    |   movel([0.402308, -0.603940, -2.826285, -1.282164, 1.570796, 1.973104],accel_mss,speed_ms,0,blend_radius_m)
    |   movel([0.405930, -0.602202, -2.826422, -1.283765, 1.570796, 1.976727],accel_mss,speed_ms,0,blend_radius_m)
    |   movel([0.409236, -0.601189, -2.826501, -1.284699, 1.570796, 1.980032],accel_mss,speed_ms,0,blend_radius_m)
    |   movel([0.412170, -0.600886, -2.826525, -1.284978, 1.570796, 1.982967],accel_mss,speed_ms,0,blend_radius_m)
    |   movel([0.414677, -0.601290, -2.826494, -1.284605, 1.570796, 1.985473],accel_mss,speed_ms,0,blend_radius_m)
    |   movel([0.416713, -0.602370, -2.826409, -1.283610, 1.570796, 1.987509],accel_mss,speed_ms,0,blend_radius_m)
    |   movel([0.418227, -0.604116, -2.826271, -1.282003, 1.570796, 1.989024],accel_mss,speed_ms,0,blend_radius_m)
    |   movel([0.419169, -0.606504, -2.826080, -1.279805, 1.570796, 1.989965],accel_mss,speed_ms,0,blend_radius_m)
    |   movel([0.419507, -0.609503, -2.825837, -1.277049, 1.570796, 1.990303],accel_mss,speed_ms,0,blend_radius_m)
    |   speed_ms = 0.005
    |   movel([0.419507, -0.603604, -2.819016, -1.289768, 1.570796, 1.990303],accel_mss,speed_ms,0,blend_radius_m)
    |   speed_ms = 0.040
    |   movel([0.367133, -0.571000, -2.821459, -1.319930, 1.570796, 1.937929],accel_mss,speed_ms,0,blend_radius_m)
    |   speed_ms = 0.005
    |   movel([0.367133, -0.576329, -2.828331, -1.307729, 1.570796, 1.937929],accel_mss,speed_ms,0,blend_radius_m)
    |   speed_ms = 0.025
    |   movel([0.368594, -0.576617, -2.828311, -1.307461, 1.570796, 1.939390],accel_mss,speed_ms,0,blend_radius_m)
    |   movel([0.369540, -0.577566, -2.828246, -1.306577, 1.570796, 1.940337],accel_mss,speed_ms,0,blend_radius_m)
    |   movel([0.369616, -0.578487, -2.828182, -1.305720, 1.570796, 1.940412],accel_mss,speed_ms,0,blend_radius_m)
    |   movel([0.369337, -0.579700, -2.828097, -1.304592, 1.570796, 1.940133],accel_mss,speed_ms,0,blend_radius_m)
    |   movel([0.368717, -0.581070, -2.828000, -1.303319, 1.570796, 1.939513],accel_mss,speed_ms,0,blend_radius_m)
    |   movel([0.367757, -0.582464, -2.827901, -1.302024, 1.570796, 1.938554],accel_mss,speed_ms,0,blend_radius_m)
    |   movel([0.365671, -0.584790, -2.827735, -1.299864, 1.570796, 1.936467],accel_mss,speed_ms,0,blend_radius_m)
    |   movel([0.364856, -0.586105, -2.827639, -1.298645, 1.570796, 1.935652],accel_mss,speed_ms,0,blend_radius_m)
    |   movel([0.364407, -0.587333, -2.827550, -1.297506, 1.570796, 1.935203],accel_mss,speed_ms,0,blend_radius_m)
    |   movel([0.364314, -0.589341, -2.827403, -1.295646, 1.570796, 1.935110],accel_mss,speed_ms,0,blend_radius_m)
    |   movel([0.364860, -0.591067, -2.827275, -1.294047, 1.570796, 1.935656],accel_mss,speed_ms,0,blend_radius_m)
    |   movel([0.365794, -0.592354, -2.827178, -1.292856, 1.570796, 1.936590],accel_mss,speed_ms,0,blend_radius_m)
    |   movel([0.367088, -0.593198, -2.827115, -1.292076, 1.570796, 1.937884],accel_mss,speed_ms,0,blend_radius_m)
    |   movel([0.368715, -0.593567, -2.827087, -1.291734, 1.570796, 1.939512],accel_mss,speed_ms,0,blend_radius_m)
    |   movel([0.366876, -0.596507, -2.826864, -1.289018, 1.570796, 1.937672],accel_mss,speed_ms,0,blend_radius_m)
    |   movel([0.365400, -0.599354, -2.826644, -1.286390, 1.570796, 1.936197],accel_mss,speed_ms,0,blend_radius_m)
    |   movel([0.364245, -0.602108, -2.826429, -1.283852, 1.570796, 1.935041],accel_mss,speed_ms,0,blend_radius_m)
    |   movel([0.363369, -0.604758, -2.826220, -1.281412, 1.570796, 1.934166],accel_mss,speed_ms,0,blend_radius_m)
    |   movel([0.362308, -0.609715, -2.825820, -1.276854, 1.570796, 1.933104],accel_mss,speed_ms,0,blend_radius_m)
    |   movel([0.361927, -0.614158, -2.825454, -1.272778, 1.570796, 1.932724],accel_mss,speed_ms,0,blend_radius_m)
    |   movel([0.361646, -0.618378, -2.825099, -1.268912, 1.570796, 1.932442],accel_mss,speed_ms,0,blend_radius_m)
    |   movel([0.361180, -0.620703, -2.824900, -1.266786, 1.570796, 1.931976],accel_mss,speed_ms,0,blend_radius_m)
    |   movel([0.360296, -0.623272, -2.824678, -1.264439, 1.570796, 1.931092],accel_mss,speed_ms,0,blend_radius_m)
    |   movel([0.358808, -0.626113, -2.824430, -1.261847, 1.570796, 1.929605],accel_mss,speed_ms,0,blend_radius_m)
    |   movel([0.356822, -0.628911, -2.824182, -1.259296, 1.570796, 1.927618],accel_mss,speed_ms,0,blend_radius_m)
    |   movel([0.354611, -0.631231, -2.823974, -1.257183, 1.570796, 1.925407],accel_mss,speed_ms,0,blend_radius_m)
    |   movel([0.352461, -0.632627, -2.823848, -1.255913, 1.570796, 1.923258],accel_mss,speed_ms,0,blend_radius_m)
    |   movel([0.353015, -0.634018, -2.823722, -1.254649, 1.570796, 1.923811],accel_mss,speed_ms,0,blend_radius_m)
    |   movel([0.353232, -0.637667, -2.823387, -1.251336, 1.570796, 1.924028],accel_mss,speed_ms,0,blend_radius_m)
    |   movel([0.352907, -0.639851, -2.823184, -1.249354, 1.570796, 1.923703],accel_mss,speed_ms,0,blend_radius_m)
    |   movel([0.351453, -0.644729, -2.822723, -1.244937, 1.570796, 1.922249],accel_mss,speed_ms,0,blend_radius_m)
    |   movel([0.350339, -0.647346, -2.822472, -1.242571, 1.570796, 1.921135],accel_mss,speed_ms,0,blend_radius_m)
    |   movel([0.348974, -0.650037, -2.822211, -1.240141, 1.570796, 1.919770],accel_mss,speed_ms,0,blend_radius_m)
    |   speed_ms = 0.005
    |   movel([0.348974, -0.643483, -2.815463, -1.253443, 1.570796, 1.919770],accel_mss,speed_ms,0,blend_radius_m)
    |   speed_ms = 0.040
    |   movel([0.338843, -0.648119, -2.815009, -1.249261, 1.570796, 1.909639],accel_mss,speed_ms,0,blend_radius_m)
    |   speed_ms = 0.005
    |   movel([0.338843, -0.654746, -2.821747, -1.235896, 1.570796, 1.909639],accel_mss,speed_ms,0,blend_radius_m)
    |   speed_ms = 0.025
    |   movel([0.341191, -0.672764, -2.819888, -1.219737, 1.570796, 1.911987],accel_mss,speed_ms,0,blend_radius_m)
    |   movel([0.341193, -0.675205, -2.819625, -1.217559, 1.570796, 1.911989],accel_mss,speed_ms,0,blend_radius_m)
    |   movel([0.340796, -0.676644, -2.819469, -1.216275, 1.570796, 1.911593],accel_mss,speed_ms,0,blend_radius_m)
    |   movel([0.339964, -0.678224, -2.819297, -1.214867, 1.570796, 1.910761],accel_mss,speed_ms,0,blend_radius_m)
    |   movel([0.337481, -0.681582, -2.818928, -1.211878, 1.570796, 1.908277],accel_mss,speed_ms,0,blend_radius_m)
    |   movel([0.336864, -0.683225, -2.818746, -1.210418, 1.570796, 1.907661],accel_mss,speed_ms,0,blend_radius_m)
    |   movel([0.336819, -0.684555, -2.818597, -1.209237, 1.570796, 1.907615],accel_mss,speed_ms,0,blend_radius_m)
    |   movel([0.337450, -0.686133, -2.818420, -1.207836, 1.570796, 1.908246],accel_mss,speed_ms,0,blend_radius_m)
    |   movel([0.338671, -0.687133, -2.818307, -1.206949, 1.570796, 1.909467],accel_mss,speed_ms,0,blend_radius_m)
    |   movel([0.341481, -0.688557, -2.818146, -1.205686, 1.570796, 1.912277],accel_mss,speed_ms,0,blend_radius_m)
    |   movel([0.342858, -0.690102, -2.817970, -1.204317, 1.570796, 1.913655],accel_mss,speed_ms,0,blend_radius_m)
    |   movel([0.344241, -0.692917, -2.817646, -1.201826, 1.570796, 1.915038],accel_mss,speed_ms,0,blend_radius_m)
    |   movel([0.344493, -0.694532, -2.817459, -1.200397, 1.570796, 1.915290],accel_mss,speed_ms,0,blend_radius_m)
    |   movel([0.344236, -0.696132, -2.817273, -1.198984, 1.570796, 1.915033],accel_mss,speed_ms,0,blend_radius_m)
    |   movel([0.343860, -0.696890, -2.817184, -1.198315, 1.570796, 1.914657],accel_mss,speed_ms,0,blend_radius_m)
    |   movel([0.343290, -0.697601, -2.817101, -1.197687, 1.570796, 1.914087],accel_mss,speed_ms,0,blend_radius_m)
    |   movel([0.341482, -0.698845, -2.816954, -1.196590, 1.570796, 1.912278],accel_mss,speed_ms,0,blend_radius_m)
    |   movel([0.341411, -0.700428, -2.816767, -1.195194, 1.570796, 1.912208],accel_mss,speed_ms,0,blend_radius_m)
    |   movel([0.341805, -0.701849, -2.816597, -1.193942, 1.570796, 1.912601],accel_mss,speed_ms,0,blend_radius_m)
    |   movel([0.343551, -0.704211, -2.816314, -1.191864, 1.570796, 1.914347],accel_mss,speed_ms,0,blend_radius_m)
    |   movel([0.347880, -0.707172, -2.815955, -1.189261, 1.570796, 1.918676],accel_mss,speed_ms,0,blend_radius_m)
    |   movel([0.350537, -0.707948, -2.815861, -1.188580, 1.570796, 1.921334],accel_mss,speed_ms,0,blend_radius_m)
    |   movel([0.353591, -0.708352, -2.815812, -1.188225, 1.570796, 1.924387],accel_mss,speed_ms,0,blend_radius_m)
    |   movel([0.356222, -0.709277, -2.815698, -1.187414, 1.570796, 1.927019],accel_mss,speed_ms,0,blend_radius_m)
    |   movel([0.357125, -0.710205, -2.815584, -1.186600, 1.570796, 1.927922],accel_mss,speed_ms,0,blend_radius_m)
    |   movel([0.357618, -0.711589, -2.815414, -1.185387, 1.570796, 1.928414],accel_mss,speed_ms,0,blend_radius_m)
    |   movel([0.357593, -0.712558, -2.815293, -1.184537, 1.570796, 1.928389],accel_mss,speed_ms,0,blend_radius_m)
    |   movel([0.357273, -0.713718, -2.815149, -1.183522, 1.570796, 1.928070],accel_mss,speed_ms,0,blend_radius_m)
    |   movel([0.356670, -0.714860, -2.815006, -1.182522, 1.570796, 1.927467],accel_mss,speed_ms,0,blend_radius_m)
    |   movel([0.355782, -0.715776, -2.814892, -1.181721, 1.570796, 1.926579],accel_mss,speed_ms,0,blend_radius_m)
    |   movel([0.354440, -0.716164, -2.814843, -1.181382, 1.570796, 1.925237],accel_mss,speed_ms,0,blend_radius_m)
    |   movel([0.349203, -0.715563, -2.814918, -1.181908, 1.570796, 1.919999],accel_mss,speed_ms,0,blend_radius_m)
    |   movel([0.344633, -0.713927, -2.815123, -1.183339, 1.570796, 1.915430],accel_mss,speed_ms,0,blend_radius_m)
    |   movel([0.344030, -0.715213, -2.814962, -1.182213, 1.570796, 1.914826],accel_mss,speed_ms,0,blend_radius_m)
    |   movel([0.343689, -0.716395, -2.814814, -1.181180, 1.570796, 1.914486],accel_mss,speed_ms,0,blend_radius_m)
    |   movel([0.343697, -0.718463, -2.814553, -1.179373, 1.570796, 1.914493],accel_mss,speed_ms,0,blend_radius_m)
    |   movel([0.344441, -0.720163, -2.814337, -1.177889, 1.570796, 1.915238],accel_mss,speed_ms,0,blend_radius_m)
    |   movel([0.345698, -0.721557, -2.814158, -1.176674, 1.570796, 1.916494],accel_mss,speed_ms,0,blend_radius_m)
    |   movel([0.348943, -0.723539, -2.813903, -1.174947, 1.570796, 1.919739],accel_mss,speed_ms,0,blend_radius_m)
    |   movel([0.351761, -0.724708, -2.813752, -1.173929, 1.570796, 1.922558],accel_mss,speed_ms,0,blend_radius_m)
    |   movel([0.352666, -0.725330, -2.813672, -1.173387, 1.570796, 1.923462],accel_mss,speed_ms,0,blend_radius_m)
    |   movel([0.352850, -0.725902, -2.813597, -1.172890, 1.570796, 1.923647],accel_mss,speed_ms,0,blend_radius_m)
    |   movel([0.352704, -0.726735, -2.813489, -1.172166, 1.570796, 1.923501],accel_mss,speed_ms,0,blend_radius_m)
    |   movel([0.352198, -0.727778, -2.813352, -1.171259, 1.570796, 1.922994],accel_mss,speed_ms,0,blend_radius_m)
    |   movel([0.351586, -0.728539, -2.813253, -1.170597, 1.570796, 1.922382],accel_mss,speed_ms,0,blend_radius_m)
    |   movel([0.350182, -0.729503, -2.813126, -1.169760, 1.570796, 1.920979],accel_mss,speed_ms,0,blend_radius_m)
    |   movel([0.348239, -0.730639, -2.812976, -1.168774, 1.570796, 1.919035],accel_mss,speed_ms,0,blend_radius_m)
    |   movel([0.347795, -0.731218, -2.812899, -1.168272, 1.570796, 1.918591],accel_mss,speed_ms,0,blend_radius_m)
    |   movel([0.347475, -0.732077, -2.812785, -1.167527, 1.570796, 1.918272],accel_mss,speed_ms,0,blend_radius_m)
    |   movel([0.347450, -0.732856, -2.812681, -1.166851, 1.570796, 1.918246],accel_mss,speed_ms,0,blend_radius_m)
    |   movel([0.348020, -0.734168, -2.812506, -1.165715, 1.570796, 1.918817],accel_mss,speed_ms,0,blend_radius_m)
    |   movel([0.349767, -0.735900, -2.812273, -1.164216, 1.570796, 1.920563],accel_mss,speed_ms,0,blend_radius_m)
    |   movel([0.358098, -0.742064, -2.811434, -1.158891, 1.570796, 1.928895],accel_mss,speed_ms,0,blend_radius_m)
    |   movel([0.358752, -0.742913, -2.811317, -1.158158, 1.570796, 1.929548],accel_mss,speed_ms,0,blend_radius_m)
    |   movel([0.359088, -0.744094, -2.811154, -1.157141, 1.570796, 1.929884],accel_mss,speed_ms,0,blend_radius_m)
    |   movel([0.358896, -0.745566, -2.810950, -1.155873, 1.570796, 1.929692],accel_mss,speed_ms,0,blend_radius_m)
    |   movel([0.357966, -0.747279, -2.810711, -1.154400, 1.570796, 1.928763],accel_mss,speed_ms,0,blend_radius_m)
    |   movel([0.356641, -0.748610, -2.810524, -1.153255, 1.570796, 1.927438],accel_mss,speed_ms,0,blend_radius_m)
    |   movel([0.355296, -0.749300, -2.810427, -1.152662, 1.570796, 1.926093],accel_mss,speed_ms,0,blend_radius_m)
    |   movel([0.354031, -0.749499, -2.810399, -1.152491, 1.570796, 1.924828],accel_mss,speed_ms,0,blend_radius_m)
    |   movel([0.352947, -0.749370, -2.810417, -1.152602, 1.570796, 1.923743],accel_mss,speed_ms,0,blend_radius_m)
    |   movel([0.347194, -0.747590, -2.810667, -1.154132, 1.570796, 1.917990],accel_mss,speed_ms,0,blend_radius_m)
    |   movel([0.341743, -0.745355, -2.810979, -1.156055, 1.570796, 1.912539],accel_mss,speed_ms,0,blend_radius_m)
    |   movel([0.336598, -0.742667, -2.811351, -1.158371, 1.570796, 1.907395],accel_mss,speed_ms,0,blend_radius_m)
    |   movel([0.331781, -0.739517, -2.811783, -1.161089, 1.570796, 1.902578],accel_mss,speed_ms,0,blend_radius_m)
    |   movel([0.330145, -0.738157, -2.811968, -1.162264, 1.570796, 1.900942],accel_mss,speed_ms,0,blend_radius_m)
    |   movel([0.328952, -0.736277, -2.812223, -1.163890, 1.570796, 1.899749],accel_mss,speed_ms,0,blend_radius_m)
    |   movel([0.328608, -0.734790, -2.812423, -1.165176, 1.570796, 1.899404],accel_mss,speed_ms,0,blend_radius_m)
    |   movel([0.328493, -0.733092, -2.812650, -1.166647, 1.570796, 1.899290],accel_mss,speed_ms,0,blend_radius_m)
    |   movel([0.328672, -0.729329, -2.813149, -1.169911, 1.570796, 1.899468],accel_mss,speed_ms,0,blend_radius_m)
    |   movel([0.330690, -0.714772, -2.815017, -1.182599, 1.570796, 1.901486],accel_mss,speed_ms,0,blend_radius_m)
    |   movel([0.330888, -0.710909, -2.815498, -1.185983, 1.570796, 1.901685],accel_mss,speed_ms,0,blend_radius_m)
    |   movel([0.330603, -0.707779, -2.815882, -1.188729, 1.570796, 1.901399],accel_mss,speed_ms,0,blend_radius_m)
    |   movel([0.330218, -0.706624, -2.816022, -1.189743, 1.570796, 1.901014],accel_mss,speed_ms,0,blend_radius_m)
    |   movel([0.329641, -0.705806, -2.816121, -1.190462, 1.570796, 1.900438],accel_mss,speed_ms,0,blend_radius_m)
    |   movel([0.328850, -0.705386, -2.816172, -1.190830, 1.570796, 1.899646],accel_mss,speed_ms,0,blend_radius_m)
    |   movel([0.327823, -0.705408, -2.816170, -1.190811, 1.570796, 1.898620],accel_mss,speed_ms,0,blend_radius_m)
    |   movel([0.325725, -0.706149, -2.816080, -1.190160, 1.570796, 1.896521],accel_mss,speed_ms,0,blend_radius_m)
    |   movel([0.324776, -0.706363, -2.816054, -1.189972, 1.570796, 1.895572],accel_mss,speed_ms,0,blend_radius_m)
    |   movel([0.324109, -0.706133, -2.816082, -1.190175, 1.570796, 1.894905],accel_mss,speed_ms,0,blend_radius_m)
    |   movel([0.323920, -0.704858, -2.816236, -1.191295, 1.570796, 1.894717],accel_mss,speed_ms,0,blend_radius_m)
    |   movel([0.324367, -0.703032, -2.816456, -1.192901, 1.570796, 1.895163],accel_mss,speed_ms,0,blend_radius_m)
    |   movel([0.326041, -0.697037, -2.817167, -1.198185, 1.570796, 1.896838],accel_mss,speed_ms,0,blend_radius_m)
    |   movel([0.327377, -0.691252, -2.817838, -1.203298, 1.570796, 1.898173],accel_mss,speed_ms,0,blend_radius_m)
    |   movel([0.329205, -0.680192, -2.819082, -1.213116, 1.570796, 1.900001],accel_mss,speed_ms,0,blend_radius_m)
    |   movel([0.330234, -0.669562, -2.820228, -1.222599, 1.570796, 1.901030],accel_mss,speed_ms,0,blend_radius_m)
    |   movel([0.330846, -0.659076, -2.821312, -1.232001, 1.570796, 1.901642],accel_mss,speed_ms,0,blend_radius_m)
    |   speed_ms = 0.005
    |   movel([0.330846, -0.652382, -2.814583, -1.245424, 1.570796, 1.901642],accel_mss,speed_ms,0,blend_radius_m)
    |   speed_ms = 0.040
    |   movel([0.322302, -0.672249, -2.812498, -1.227642, 1.570796, 1.893098],accel_mss,speed_ms,0,blend_radius_m)
    |   speed_ms = 0.005
    |   movel([0.322302, -0.679246, -2.819186, -1.213958, 1.570796, 1.893098],accel_mss,speed_ms,0,blend_radius_m)
    |   speed_ms = 0.025
    |   movel([0.317406, -0.692411, -2.817705, -1.202273, 1.570796, 1.888202],accel_mss,speed_ms,0,blend_radius_m)
    |   movel([0.314679, -0.699052, -2.816930, -1.196407, 1.570796, 1.885475],accel_mss,speed_ms,0,blend_radius_m)
    |   movel([0.311784, -0.705705, -2.816134, -1.190550, 1.570796, 1.882580],accel_mss,speed_ms,0,blend_radius_m)
    |   movel([0.309555, -0.704357, -2.816297, -1.191736, 1.570796, 1.880351],accel_mss,speed_ms,0,blend_radius_m)
    |   movel([0.309119, -0.704207, -2.816315, -1.191868, 1.570796, 1.879915],accel_mss,speed_ms,0,blend_radius_m)
    |   movel([0.308518, -0.704441, -2.816286, -1.191661, 1.570796, 1.879314],accel_mss,speed_ms,0,blend_radius_m)
    |   movel([0.307864, -0.705178, -2.816197, -1.191013, 1.570796, 1.878660],accel_mss,speed_ms,0,blend_radius_m)
    |   movel([0.307348, -0.706068, -2.816090, -1.190231, 1.570796, 1.878144],accel_mss,speed_ms,0,blend_radius_m)
    |   movel([0.304158, -0.711556, -2.815418, -1.185415, 1.570796, 1.874954],accel_mss,speed_ms,0,blend_radius_m)
    |   movel([0.300492, -0.716914, -2.814749, -1.180727, 1.570796, 1.871289],accel_mss,speed_ms,0,blend_radius_m)
    |   movel([0.299529, -0.718081, -2.814601, -1.179707, 1.570796, 1.870325],accel_mss,speed_ms,0,blend_radius_m)
    |   movel([0.298588, -0.718738, -2.814518, -1.179133, 1.570796, 1.869384],accel_mss,speed_ms,0,blend_radius_m)
    |   movel([0.298139, -0.718483, -2.814550, -1.179356, 1.570796, 1.868936],accel_mss,speed_ms,0,blend_radius_m)
    |   movel([0.298067, -0.717756, -2.814642, -1.179991, 1.570796, 1.868864],accel_mss,speed_ms,0,blend_radius_m)
    |   movel([0.298588, -0.712578, -2.815291, -1.184520, 1.570796, 1.869384],accel_mss,speed_ms,0,blend_radius_m)
    |   movel([0.299943, -0.706821, -2.815998, -1.189570, 1.570796, 1.870739],accel_mss,speed_ms,0,blend_radius_m)
    |   speed_ms = 0.005
    |   movel([0.299943, -0.699432, -2.809373, -1.203585, 1.570796, 1.870739],accel_mss,speed_ms,0,blend_radius_m)
    |   speed_ms = 0.040
    |   movel([0.306015, -0.706814, -2.808468, -1.197107, 1.570796, 1.876811],accel_mss,speed_ms,0,blend_radius_m)
    |   speed_ms = 0.005
    |   movel([0.306015, -0.714306, -2.815076, -1.183007, 1.570796, 1.876811],accel_mss,speed_ms,0,blend_radius_m)
    |   speed_ms = 0.025
    |   movel([0.304087, -0.722707, -2.814011, -1.175672, 1.570796, 1.874884],accel_mss,speed_ms,0,blend_radius_m)
    |   movel([0.302756, -0.727093, -2.813442, -1.171854, 1.570796, 1.873552],accel_mss,speed_ms,0,blend_radius_m)
    |   movel([0.299423, -0.736108, -2.812245, -1.164036, 1.570796, 1.870219],accel_mss,speed_ms,0,blend_radius_m)
    |   movel([0.297435, -0.740698, -2.811622, -1.160069, 1.570796, 1.868232],accel_mss,speed_ms,0,blend_radius_m)
    |   movel([0.292872, -0.749937, -2.810337, -1.152115, 1.570796, 1.863668],accel_mss,speed_ms,0,blend_radius_m)
    |   movel([0.293684, -0.747094, -2.810737, -1.154559, 1.570796, 1.864480],accel_mss,speed_ms,0,blend_radius_m)
    |   movel([0.293813, -0.744675, -2.811074, -1.156641, 1.570796, 1.864609],accel_mss,speed_ms,0,blend_radius_m)
    |   movel([0.293266, -0.742844, -2.811327, -1.158218, 1.570796, 1.864063],accel_mss,speed_ms,0,blend_radius_m)
    |   movel([0.292050, -0.741767, -2.811475, -1.159147, 1.570796, 1.862846],accel_mss,speed_ms,0,blend_radius_m)
    |   speed_ms = 0.005
    |   movel([0.292050, -0.733915, -2.804935, -1.173539, 1.570796, 1.862846],accel_mss,speed_ms,0,blend_radius_m)
    |   speed_ms = 0.040
    |   movel([0.264567, -0.752845, -2.802266, -1.157279, 1.570796, 1.835363],accel_mss,speed_ms,0,blend_radius_m)
    |   speed_ms = 0.005
    |   movel([0.264567, -0.760932, -2.808755, -1.142701, 1.570796, 1.835363],accel_mss,speed_ms,0,blend_radius_m)
    |   speed_ms = 0.025
    |   movel([0.259716, -0.767291, -2.807814, -1.137284, 1.570796, 1.830512],accel_mss,speed_ms,0,blend_radius_m)
    |   movel([0.254573, -0.773267, -2.806912, -1.132211, 1.570796, 1.825369],accel_mss,speed_ms,0,blend_radius_m)
    |   movel([0.249228, -0.778773, -2.806065, -1.127552, 1.570796, 1.820024],accel_mss,speed_ms,0,blend_radius_m)
    |   movel([0.243766, -0.783719, -2.805291, -1.123379, 1.570796, 1.814562],accel_mss,speed_ms,0,blend_radius_m)
    |   movel([0.245185, -0.780912, -2.805732, -1.125745, 1.570796, 1.815981],accel_mss,speed_ms,0,blend_radius_m)
    |   movel([0.246261, -0.778308, -2.806137, -1.127944, 1.570796, 1.817058],accel_mss,speed_ms,0,blend_radius_m)
    |   movel([0.246914, -0.776137, -2.806472, -1.129780, 1.570796, 1.817711],accel_mss,speed_ms,0,blend_radius_m)
    |   movel([0.247067, -0.774630, -2.806703, -1.131056, 1.570796, 1.817864],accel_mss,speed_ms,0,blend_radius_m)
    |   movel([0.246632, -0.774034, -2.806795, -1.131561, 1.570796, 1.817428],accel_mss,speed_ms,0,blend_radius_m)
    |   movel([0.246172, -0.774146, -2.806777, -1.131465, 1.570796, 1.816969],accel_mss,speed_ms,0,blend_radius_m)
    |   movel([0.245530, -0.774575, -2.806712, -1.131102, 1.570796, 1.816326],accel_mss,speed_ms,0,blend_radius_m)
    |   movel([0.243691, -0.776486, -2.806418, -1.129484, 1.570796, 1.814487],accel_mss,speed_ms,0,blend_radius_m)
    |   movel([0.238993, -0.782767, -2.805441, -1.124181, 1.570796, 1.809789],accel_mss,speed_ms,0,blend_radius_m)
    |   movel([0.236811, -0.785491, -2.805011, -1.121887, 1.570796, 1.807608],accel_mss,speed_ms,0,blend_radius_m)
    |   movel([0.232164, -0.790621, -2.804191, -1.117576, 1.570796, 1.802960],accel_mss,speed_ms,0,blend_radius_m)
    |   movel([0.229754, -0.792963, -2.803813, -1.115614, 1.570796, 1.800550],accel_mss,speed_ms,0,blend_radius_m)
    |   movel([0.227322, -0.795102, -2.803464, -1.113822, 1.570796, 1.798118],accel_mss,speed_ms,0,blend_radius_m)
    |   movel([0.224892, -0.797019, -2.803150, -1.112220, 1.570796, 1.795689],accel_mss,speed_ms,0,blend_radius_m)
    |   movel([0.222500, -0.798662, -2.802879, -1.110847, 1.570796, 1.793297],accel_mss,speed_ms,0,blend_radius_m)
    |   movel([0.225551, -0.794203, -2.803611, -1.114575, 1.570796, 1.796348],accel_mss,speed_ms,0,blend_radius_m)
    |   movel([0.228539, -0.789683, -2.804342, -1.118364, 1.570796, 1.799335],accel_mss,speed_ms,0,blend_radius_m)
    |   movel([0.229939, -0.786753, -2.804811, -1.120825, 1.570796, 1.800735],accel_mss,speed_ms,0,blend_radius_m)
    |   movel([0.230766, -0.784004, -2.805246, -1.123139, 1.570796, 1.801562],accel_mss,speed_ms,0,blend_radius_m)
    |   movel([0.230727, -0.783146, -2.805382, -1.123862, 1.570796, 1.801524],accel_mss,speed_ms,0,blend_radius_m)
    |   movel([0.230255, -0.782877, -2.805424, -1.124088, 1.570796, 1.801051],accel_mss,speed_ms,0,blend_radius_m)
    |   movel([0.229262, -0.783376, -2.805345, -1.123668, 1.570796, 1.800059],accel_mss,speed_ms,0,blend_radius_m)
    |   movel([0.227654, -0.784825, -2.805117, -1.122447, 1.570796, 1.798450],accel_mss,speed_ms,0,blend_radius_m)
    |   movel([0.219165, -0.793679, -2.803696, -1.115014, 1.570796, 1.789962],accel_mss,speed_ms,0,blend_radius_m)
    |   movel([0.214935, -0.797579, -2.803058, -1.111752, 1.570796, 1.785731],accel_mss,speed_ms,0,blend_radius_m)
    |   movel([0.212831, -0.799195, -2.802791, -1.110402, 1.570796, 1.783628],accel_mss,speed_ms,0,blend_radius_m)
    |   movel([0.210731, -0.800519, -2.802572, -1.109298, 1.570796, 1.781527],accel_mss,speed_ms,0,blend_radius_m)
    |   speed_ms = 0.005
    |   movel([0.210731, -0.791984, -2.796194, -1.124210, 1.570796, 1.781527],accel_mss,speed_ms,0,blend_radius_m)
    |   speed_ms = 0.040
    |   movel([0.250936, -0.732671, -2.805105, -1.174613, 1.570796, 1.821733],accel_mss,speed_ms,0,blend_radius_m)
    |   speed_ms = 0.005
    |   movel([0.250936, -0.740507, -2.811648, -1.160234, 1.570796, 1.821733],accel_mss,speed_ms,0,blend_radius_m)
    |   speed_ms = 0.025
    |   movel([0.251221, -0.737209, -2.812097, -1.163083, 1.570796, 1.822018],accel_mss,speed_ms,0,blend_radius_m)
    |   movel([0.252157, -0.733520, -2.812593, -1.166276, 1.570796, 1.822953],accel_mss,speed_ms,0,blend_radius_m)
    |   movel([0.253672, -0.729520, -2.813124, -1.169746, 1.570796, 1.824469],accel_mss,speed_ms,0,blend_radius_m)
    |   movel([0.255690, -0.725314, -2.813674, -1.173401, 1.570796, 1.826486],accel_mss,speed_ms,0,blend_radius_m)
    |   movel([0.258152, -0.720982, -2.814232, -1.177175, 1.570796, 1.828949],accel_mss,speed_ms,0,blend_radius_m)
    |   movel([0.260973, -0.716636, -2.814784, -1.180970, 1.570796, 1.831770],accel_mss,speed_ms,0,blend_radius_m)
    |   movel([0.264090, -0.712359, -2.815318, -1.184712, 1.570796, 1.834886],accel_mss,speed_ms,0,blend_radius_m)
    |   movel([0.267414, -0.708265, -2.815822, -1.188302, 1.570796, 1.838210],accel_mss,speed_ms,0,blend_radius_m)
    |   movel([0.271698, -0.703495, -2.816400, -1.192494, 1.570796, 1.842494],accel_mss,speed_ms,0,blend_radius_m)
    |   movel([0.280462, -0.694106, -2.817509, -1.200774, 1.570796, 1.851259],accel_mss,speed_ms,0,blend_radius_m)
    |   movel([0.284726, -0.689132, -2.818081, -1.205176, 1.570796, 1.855522],accel_mss,speed_ms,0,blend_radius_m)
    |   movel([0.288727, -0.683680, -2.818695, -1.210014, 1.570796, 1.859523],accel_mss,speed_ms,0,blend_radius_m)
    |   movel([0.290511, -0.680842, -2.819010, -1.212537, 1.570796, 1.861308],accel_mss,speed_ms,0,blend_radius_m)
    |   movel([0.292070, -0.678025, -2.819319, -1.215045, 1.570796, 1.862866],accel_mss,speed_ms,0,blend_radius_m)
    |   movel([0.293342, -0.675299, -2.819615, -1.217475, 1.570796, 1.864138],accel_mss,speed_ms,0,blend_radius_m)
    |   movel([0.294269, -0.672734, -2.819891, -1.219764, 1.570796, 1.865066],accel_mss,speed_ms,0,blend_radius_m)
    |   movel([0.294776, -0.670420, -2.820137, -1.221832, 1.570796, 1.865573],accel_mss,speed_ms,0,blend_radius_m)
    |   movel([0.294799, -0.668431, -2.820347, -1.223611, 1.570796, 1.865595],accel_mss,speed_ms,0,blend_radius_m)
    |   speed_ms = 0.005
    |   movel([0.294799, -0.661596, -2.813637, -1.237157, 1.570796, 1.865595],accel_mss,speed_ms,0,blend_radius_m)
    |   speed_ms = 0.040
    |   movel([0.293952, -0.646497, -2.815169, -1.250724, 1.570796, 1.864749],accel_mss,speed_ms,0,blend_radius_m)
    |   speed_ms = 0.005
    |   movel([0.293952, -0.653098, -2.821910, -1.237381, 1.570796, 1.864749],accel_mss,speed_ms,0,blend_radius_m)
    |   speed_ms = 0.025
    |   movel([0.289382, -0.667550, -2.820440, -1.224399, 1.570796, 1.860178],accel_mss,speed_ms,0,blend_radius_m)
    |   movel([0.287826, -0.670954, -2.820080, -1.221354, 1.570796, 1.858622],accel_mss,speed_ms,0,blend_radius_m)
    |   movel([0.285585, -0.674371, -2.819715, -1.218302, 1.570796, 1.856381],accel_mss,speed_ms,0,blend_radius_m)
    |   movel([0.282917, -0.677576, -2.819368, -1.215445, 1.570796, 1.853713],accel_mss,speed_ms,0,blend_radius_m)
    |   movel([0.274021, -0.687068, -2.818315, -1.207007, 1.570796, 1.844818],accel_mss,speed_ms,0,blend_radius_m)
    |   movel([0.271013, -0.690670, -2.817905, -1.203814, 1.570796, 1.841809],accel_mss,speed_ms,0,blend_radius_m)
    |   movel([0.268158, -0.694394, -2.817475, -1.200519, 1.570796, 1.838955],accel_mss,speed_ms,0,blend_radius_m)
    |   movel([0.265483, -0.698194, -2.817031, -1.197164, 1.570796, 1.836279],accel_mss,speed_ms,0,blend_radius_m)
    |   movel([0.263207, -0.701950, -2.816585, -1.193854, 1.570796, 1.834004],accel_mss,speed_ms,0,blend_radius_m)
    |   movel([0.261257, -0.705686, -2.816136, -1.190567, 1.570796, 1.832054],accel_mss,speed_ms,0,blend_radius_m)
    |   movel([0.259346, -0.709389, -2.815685, -1.187315, 1.570796, 1.830143],accel_mss,speed_ms,0,blend_radius_m)
    |   movel([0.257194, -0.713055, -2.815232, -1.184102, 1.570796, 1.827990],accel_mss,speed_ms,0,blend_radius_m)
    |   movel([0.255717, -0.707028, -2.815973, -1.189388, 1.570796, 1.826513],accel_mss,speed_ms,0,blend_radius_m)
    |   movel([0.256055, -0.704871, -2.816234, -1.191283, 1.570796, 1.826852],accel_mss,speed_ms,0,blend_radius_m)
    |   movel([0.256723, -0.702568, -2.816511, -1.193310, 1.570796, 1.827519],accel_mss,speed_ms,0,blend_radius_m)
    |   movel([0.257718, -0.700113, -2.816804, -1.195472, 1.570796, 1.828514],accel_mss,speed_ms,0,blend_radius_m)
    |   movel([0.259061, -0.697485, -2.817114, -1.197790, 1.570796, 1.829857],accel_mss,speed_ms,0,blend_radius_m)
    |   movel([0.261535, -0.693777, -2.817547, -1.201065, 1.570796, 1.832331],accel_mss,speed_ms,0,blend_radius_m)
    |   movel([0.265125, -0.689223, -2.818070, -1.205096, 1.570796, 1.835921],accel_mss,speed_ms,0,blend_radius_m)
    |   movel([0.273962, -0.678865, -2.819227, -1.214297, 1.570796, 1.844758],accel_mss,speed_ms,0,blend_radius_m)
    |   movel([0.278345, -0.673728, -2.819784, -1.218876, 1.570796, 1.849141],accel_mss,speed_ms,0,blend_radius_m)
    |   movel([0.282110, -0.669069, -2.820280, -1.223040, 1.570796, 1.852906],accel_mss,speed_ms,0,blend_radius_m)
    |   movel([0.284800, -0.665246, -2.820680, -1.226463, 1.570796, 1.855596],accel_mss,speed_ms,0,blend_radius_m)
    |   movel([0.285602, -0.663751, -2.820835, -1.227803, 1.570796, 1.856398],accel_mss,speed_ms,0,blend_radius_m)
    |   movel([0.285959, -0.662596, -2.820953, -1.228839, 1.570796, 1.856756],accel_mss,speed_ms,0,blend_radius_m)
    |   speed_ms = 0.005
    |   movel([0.285959, -0.655849, -2.814231, -1.242309, 1.570796, 1.856756],accel_mss,speed_ms,0,blend_radius_m)
    |   speed_ms = 0.040
    |   movel([0.270387, -0.659389, -2.813866, -1.239133, 1.570796, 1.841184],accel_mss,speed_ms,0,blend_radius_m)
    |   speed_ms = 0.005
    |   movel([0.270387, -0.666191, -2.820582, -1.225616, 1.570796, 1.841184],accel_mss,speed_ms,0,blend_radius_m)
    |   speed_ms = 0.025
    |   movel([0.268885, -0.666508, -2.820548, -1.225332, 1.570796, 1.839682],accel_mss,speed_ms,0,blend_radius_m)
    |   movel([0.267667, -0.666361, -2.820564, -1.225464, 1.570796, 1.838463],accel_mss,speed_ms,0,blend_radius_m)
    |   movel([0.265946, -0.664969, -2.820709, -1.226712, 1.570796, 1.836743],accel_mss,speed_ms,0,blend_radius_m)
    |   movel([0.264961, -0.662550, -2.820958, -1.228881, 1.570796, 1.835757],accel_mss,speed_ms,0,blend_radius_m)
    |   movel([0.264459, -0.659627, -2.821257, -1.231506, 1.570796, 1.835256],accel_mss,speed_ms,0,blend_radius_m)
    |   movel([0.264494, -0.658384, -2.821382, -1.232623, 1.570796, 1.835291],accel_mss,speed_ms,0,blend_radius_m)
    |   movel([0.265649, -0.655850, -2.821637, -1.234902, 1.570796, 1.836445],accel_mss,speed_ms,0,blend_radius_m)
    |   movel([0.269640, -0.648483, -2.822362, -1.241544, 1.570796, 1.840436],accel_mss,speed_ms,0,blend_radius_m)
    |   movel([0.277178, -0.633658, -2.823755, -1.254976, 1.570796, 1.847974],accel_mss,speed_ms,0,blend_radius_m)
    |   movel([0.280706, -0.626236, -2.824419, -1.261734, 1.570796, 1.851502],accel_mss,speed_ms,0,blend_radius_m)
    |   speed_ms = 0.005
    |   movel([0.280706, -0.620062, -2.817627, -1.274700, 1.570796, 1.851502],accel_mss,speed_ms,0,blend_radius_m)
    |   speed_ms = 0.040
    |   movel([0.269956, -0.628365, -2.816885, -1.267138, 1.570796, 1.840752],accel_mss,speed_ms,0,blend_radius_m)
    |   speed_ms = 0.005
    |   movel([0.269956, -0.634676, -2.823662, -1.254051, 1.570796, 1.840752],accel_mss,speed_ms,0,blend_radius_m)
    |   speed_ms = 0.025
    |   movel([0.268196, -0.639015, -2.823262, -1.250112, 1.570796, 1.838992],accel_mss,speed_ms,0,blend_radius_m)
    |   movel([0.266046, -0.643470, -2.822843, -1.246077, 1.570796, 1.836843],accel_mss,speed_ms,0,blend_radius_m)
    |   movel([0.263426, -0.647851, -2.822423, -1.242115, 1.570796, 1.834223],accel_mss,speed_ms,0,blend_radius_m)
    |   movel([0.261912, -0.649965, -2.822218, -1.240206, 1.570796, 1.832708],accel_mss,speed_ms,0,blend_radius_m)
    |   movel([0.258643, -0.653989, -2.821822, -1.236578, 1.570796, 1.829439],accel_mss,speed_ms,0,blend_radius_m)
    |   movel([0.257809, -0.655756, -2.821646, -1.234987, 1.570796, 1.828605],accel_mss,speed_ms,0,blend_radius_m)
    |   movel([0.252740, -0.668890, -2.820299, -1.223201, 1.570796, 1.823536],accel_mss,speed_ms,0,blend_radius_m)
    |   movel([0.252286, -0.670142, -2.820167, -1.222081, 1.570796, 1.823082],accel_mss,speed_ms,0,blend_radius_m)
    |   movel([0.252127, -0.671193, -2.820055, -1.221141, 1.570796, 1.822924],accel_mss,speed_ms,0,blend_radius_m)
    |   movel([0.252744, -0.671921, -2.819978, -1.220490, 1.570796, 1.823541],accel_mss,speed_ms,0,blend_radius_m)
    |   movel([0.253910, -0.671947, -2.819975, -1.220467, 1.570796, 1.824706],accel_mss,speed_ms,0,blend_radius_m)
    |   movel([0.257351, -0.671833, -2.819987, -1.220569, 1.570796, 1.828147],accel_mss,speed_ms,0,blend_radius_m)
    |   movel([0.260449, -0.672279, -2.819939, -1.220171, 1.570796, 1.831245],accel_mss,speed_ms,0,blend_radius_m)
    |   movel([0.262955, -0.673536, -2.819805, -1.219048, 1.570796, 1.833751],accel_mss,speed_ms,0,blend_radius_m)
    |   movel([0.264597, -0.675872, -2.819553, -1.216963, 1.570796, 1.835393],accel_mss,speed_ms,0,blend_radius_m)
    |   speed_ms = 0.005
    |   movel([0.264597, -0.668926, -2.812858, -1.230605, 1.570796, 1.835393],accel_mss,speed_ms,0,blend_radius_m)
    |   speed_ms = 0.040
    |   movel([0.251923, -0.701660, -2.809102, -1.201627, 1.570796, 1.822719],accel_mss,speed_ms,0,blend_radius_m)
    |   speed_ms = 0.005
    |   movel([0.251923, -0.709081, -2.815722, -1.187586, 1.570796, 1.822719],accel_mss,speed_ms,0,blend_radius_m)
    |   speed_ms = 0.025
    |   movel([0.251162, -0.709883, -2.815624, -1.186882, 1.570796, 1.821958],accel_mss,speed_ms,0,blend_radius_m)
    |   movel([0.250457, -0.710871, -2.815502, -1.186016, 1.570796, 1.821253],accel_mss,speed_ms,0,blend_radius_m)
    |   movel([0.247600, -0.715898, -2.814876, -1.181615, 1.570796, 1.818396],accel_mss,speed_ms,0,blend_radius_m)
    |   movel([0.247141, -0.716386, -2.814815, -1.181188, 1.570796, 1.817938],accel_mss,speed_ms,0,blend_radius_m)
    |   movel([0.246494, -0.716647, -2.814782, -1.180960, 1.570796, 1.817290],accel_mss,speed_ms,0,blend_radius_m)
    |   movel([0.246025, -0.716409, -2.814812, -1.181168, 1.570796, 1.816821],accel_mss,speed_ms,0,blend_radius_m)
    |   movel([0.245537, -0.714935, -2.814997, -1.182457, 1.570796, 1.816333],accel_mss,speed_ms,0,blend_radius_m)
    |   movel([0.245593, -0.711455, -2.815430, -1.185504, 1.570796, 1.816389],accel_mss,speed_ms,0,blend_radius_m)
    |   movel([0.246638, -0.707577, -2.815906, -1.188906, 1.570796, 1.817435],accel_mss,speed_ms,0,blend_radius_m)
    |   movel([0.248205, -0.703406, -2.816411, -1.192572, 1.570796, 1.819002],accel_mss,speed_ms,0,blend_radius_m)
    |   movel([0.250034, -0.699181, -2.816914, -1.196294, 1.570796, 1.820830],accel_mss,speed_ms,0,blend_radius_m)
    |   movel([0.252152, -0.695004, -2.817404, -1.199981, 1.570796, 1.822948],accel_mss,speed_ms,0,blend_radius_m)
    |   movel([0.254547, -0.690879, -2.817881, -1.203629, 1.570796, 1.825343],accel_mss,speed_ms,0,blend_radius_m)
    |   movel([0.257207, -0.686805, -2.818344, -1.207239, 1.570796, 1.828003],accel_mss,speed_ms,0,blend_radius_m)
    |   movel([0.260126, -0.682780, -2.818795, -1.210814, 1.570796, 1.830922],accel_mss,speed_ms,0,blend_radius_m)
    |   movel([0.263284, -0.678810, -2.819233, -1.214345, 1.570796, 1.834080],accel_mss,speed_ms,0,blend_radius_m)
    |   movel([0.266680, -0.674885, -2.819660, -1.217844, 1.570796, 1.837476],accel_mss,speed_ms,0,blend_radius_m)
    |   movel([0.270295, -0.671014, -2.820074, -1.221301, 1.570796, 1.841091],accel_mss,speed_ms,0,blend_radius_m)
    |   movel([0.275326, -0.665239, -2.820681, -1.226469, 1.570796, 1.846122],accel_mss,speed_ms,0,blend_radius_m)
    |   movel([0.280639, -0.658479, -2.821373, -1.232538, 1.570796, 1.851436],accel_mss,speed_ms,0,blend_radius_m)
    |   movel([0.286421, -0.650648, -2.822151, -1.239590, 1.570796, 1.857218],accel_mss,speed_ms,0,blend_radius_m)
    |   speed_ms = 0.005
    |   movel([0.286421, -0.644084, -2.815405, -1.252900, 1.570796, 1.857218],accel_mss,speed_ms,0,blend_radius_m)
    |   speed_ms = 0.040
    |   movel([0.281742, -0.645946, -2.815223, -1.251220, 1.570796, 1.852539],accel_mss,speed_ms,0,blend_radius_m)
    |   speed_ms = 0.005
    |   movel([0.281742, -0.652539, -2.821966, -1.237885, 1.570796, 1.852539],accel_mss,speed_ms,0,blend_radius_m)
    |   speed_ms = 0.025
    |   movel([0.286599, -0.642016, -2.822980, -1.247392, 1.570796, 1.857395],accel_mss,speed_ms,0,blend_radius_m)
    |   movel([0.292005, -0.631247, -2.823973, -1.257169, 1.570796, 1.862802],accel_mss,speed_ms,0,blend_radius_m)
    |   movel([0.295023, -0.625810, -2.824456, -1.262123, 1.570796, 1.865819],accel_mss,speed_ms,0,blend_radius_m)
    |   movel([0.298291, -0.620365, -2.824929, -1.267095, 1.570796, 1.869087],accel_mss,speed_ms,0,blend_radius_m)
    |   movel([0.301867, -0.614919, -2.825390, -1.272080, 1.570796, 1.872663],accel_mss,speed_ms,0,blend_radius_m)
    |   movel([0.305771, -0.609511, -2.825836, -1.277042, 1.570796, 1.876568],accel_mss,speed_ms,0,blend_radius_m)
    |   movel([0.316584, -0.595902, -2.826910, -1.289577, 1.570796, 1.887381],accel_mss,speed_ms,0,blend_radius_m)
    |   movel([0.321306, -0.589653, -2.827379, -1.295356, 1.570796, 1.892102],accel_mss,speed_ms,0,blend_radius_m)
    |   movel([0.323553, -0.586451, -2.827614, -1.298324, 1.570796, 1.894350],accel_mss,speed_ms,0,blend_radius_m)
    |   movel([0.325620, -0.583188, -2.827850, -1.301351, 1.570796, 1.896416],accel_mss,speed_ms,0,blend_radius_m)
    |   movel([0.330441, -0.573450, -2.828528, -1.310410, 1.570796, 1.901237],accel_mss,speed_ms,0,blend_radius_m)
    |   speed_ms = 0.005
    |   movel([0.330441, -0.568173, -2.821652, -1.322564, 1.570796, 1.901237],accel_mss,speed_ms,0,blend_radius_m)
    |   speed_ms = 0.040
    |   movel([0.342207, -0.545734, -2.823077, -1.343579, 1.570796, 1.913003],accel_mss,speed_ms,0,blend_radius_m)
    |   speed_ms = 0.005
    |   movel([0.342207, -0.550601, -2.829983, -1.331805, 1.570796, 1.913003],accel_mss,speed_ms,0,blend_radius_m)
    |   speed_ms = 0.025
    |   movel([0.346052, -0.542532, -2.830451, -1.339405, 1.570796, 1.916848],accel_mss,speed_ms,0,blend_radius_m)
    |   movel([0.348494, -0.538436, -2.830680, -1.343273, 1.570796, 1.919290],accel_mss,speed_ms,0,blend_radius_m)
    |   movel([0.351462, -0.534417, -2.830899, -1.347073, 1.570796, 1.922258],accel_mss,speed_ms,0,blend_radius_m)
    |   movel([0.353819, -0.531799, -2.831038, -1.349551, 1.570796, 1.924616],accel_mss,speed_ms,0,blend_radius_m)
    |   movel([0.356263, -0.529422, -2.831163, -1.351804, 1.570796, 1.927060],accel_mss,speed_ms,0,blend_radius_m)
    |   movel([0.361255, -0.525041, -2.831387, -1.355961, 1.570796, 1.932051],accel_mss,speed_ms,0,blend_radius_m)
    |   movel([0.365767, -0.520752, -2.831600, -1.360038, 1.570796, 1.936563],accel_mss,speed_ms,0,blend_radius_m)
    |   movel([0.369477, -0.516480, -2.831805, -1.364104, 1.570796, 1.940273],accel_mss,speed_ms,0,blend_radius_m)
    |   movel([0.376777, -0.506547, -2.832258, -1.373584, 1.570796, 1.947573],accel_mss,speed_ms,0,blend_radius_m)
    |   movel([0.378349, -0.504567, -2.832344, -1.375478, 1.570796, 1.949145],accel_mss,speed_ms,0,blend_radius_m)
    |   movel([0.380026, -0.502771, -2.832421, -1.377197, 1.570796, 1.950823],accel_mss,speed_ms,0,blend_radius_m)
    |   movel([0.383597, -0.499591, -2.832555, -1.380243, 1.570796, 1.954394],accel_mss,speed_ms,0,blend_radius_m)
    |   movel([0.390818, -0.493833, -2.832788, -1.385768, 1.570796, 1.961615],accel_mss,speed_ms,0,blend_radius_m)
    |   movel([0.398572, -0.486986, -2.833050, -1.392353, 1.570796, 1.969369],accel_mss,speed_ms,0,blend_radius_m)
    |   movel([0.402468, -0.483224, -2.833188, -1.395978, 1.570796, 1.973265],accel_mss,speed_ms,0,blend_radius_m)
    |   movel([0.406308, -0.479074, -2.833334, -1.399981, 1.570796, 1.977105],accel_mss,speed_ms,0,blend_radius_m)
    |   movel([0.409213, -0.475357, -2.833459, -1.403573, 1.570796, 1.980009],accel_mss,speed_ms,0,blend_radius_m)
    |   movel([0.411609, -0.471549, -2.833583, -1.407257, 1.570796, 1.982406],accel_mss,speed_ms,0,blend_radius_m)
    |   movel([0.412944, -0.468362, -2.833683, -1.410344, 1.570796, 1.983740],accel_mss,speed_ms,0,blend_radius_m)
    |   movel([0.413038, -0.467231, -2.833718, -1.411441, 1.570796, 1.983834],accel_mss,speed_ms,0,blend_radius_m)
    |   movel([0.412653, -0.466529, -2.833739, -1.412121, 1.570796, 1.983450],accel_mss,speed_ms,0,blend_radius_m)
    |   movel([0.410952, -0.466142, -2.833750, -1.412497, 1.570796, 1.981749],accel_mss,speed_ms,0,blend_radius_m)
    |   movel([0.408462, -0.466641, -2.833735, -1.412012, 1.570796, 1.979258],accel_mss,speed_ms,0,blend_radius_m)
    |   movel([0.405362, -0.467913, -2.833697, -1.410779, 1.570796, 1.976159],accel_mss,speed_ms,0,blend_radius_m)
    |   movel([0.401878, -0.469798, -2.833638, -1.408952, 1.570796, 1.972675],accel_mss,speed_ms,0,blend_radius_m)
    |   movel([0.398201, -0.472185, -2.833563, -1.406641, 1.570796, 1.968997],accel_mss,speed_ms,0,blend_radius_m)
    |   movel([0.394540, -0.474917, -2.833474, -1.403998, 1.570796, 1.965337],accel_mss,speed_ms,0,blend_radius_m)
    |   movel([0.391096, -0.477871, -2.833375, -1.401143, 1.570796, 1.961892],accel_mss,speed_ms,0,blend_radius_m)
    |   movel([0.388061, -0.480910, -2.833270, -1.398209, 1.570796, 1.958858],accel_mss,speed_ms,0,blend_radius_m)
    |   movel([0.383868, -0.485988, -2.833087, -1.393313, 1.570796, 1.954664],accel_mss,speed_ms,0,blend_radius_m)
    |   movel([0.372155, -0.501536, -2.832474, -1.378379, 1.570796, 1.942951],accel_mss,speed_ms,0,blend_radius_m)
    |   movel([0.364143, -0.511496, -2.832037, -1.368856, 1.570796, 1.934940],accel_mss,speed_ms,0,blend_radius_m)
    |   movel([0.356918, -0.519535, -2.831659, -1.361195, 1.570796, 1.927714],accel_mss,speed_ms,0,blend_radius_m)
    |   movel([0.353354, -0.523432, -2.831467, -1.357490, 1.570796, 1.924150],accel_mss,speed_ms,0,blend_radius_m)
    |   movel([0.349966, -0.527467, -2.831264, -1.353659, 1.570796, 1.920762],accel_mss,speed_ms,0,blend_radius_m)
    |   movel([0.346734, -0.531828, -2.831037, -1.349524, 1.570796, 1.917530],accel_mss,speed_ms,0,blend_radius_m)
    |   movel([0.343810, -0.536199, -2.830803, -1.345387, 1.570796, 1.914606],accel_mss,speed_ms,0,blend_radius_m)
    |   movel([0.341163, -0.540567, -2.830562, -1.341260, 1.570796, 1.911959],accel_mss,speed_ms,0,blend_radius_m)
    |   movel([0.338760, -0.544901, -2.830316, -1.337172, 1.570796, 1.909556],accel_mss,speed_ms,0,blend_radius_m)
    |   movel([0.334545, -0.553403, -2.829815, -1.329171, 1.570796, 1.905341],accel_mss,speed_ms,0,blend_radius_m)
    |   movel([0.330875, -0.561563, -2.829309, -1.321517, 1.570796, 1.901671],accel_mss,speed_ms,0,blend_radius_m)
    |   speed_ms = 0.005
    |   movel([0.330875, -0.556497, -2.822417, -1.333476, 1.570796, 1.901671],accel_mss,speed_ms,0,blend_radius_m)
    |   speed_ms = 0.040
    |   movel([0.322044, -0.564451, -2.821901, -1.326037, 1.570796, 1.892840],accel_mss,speed_ms,0,blend_radius_m)
    |   speed_ms = 0.005
    |   movel([0.322044, -0.569661, -2.828783, -1.313945, 1.570796, 1.892840],accel_mss,speed_ms,0,blend_radius_m)
    |   speed_ms = 0.025
    |   movel([0.328064, -0.556756, -2.829610, -1.326023, 1.570796, 1.898861],accel_mss,speed_ms,0,blend_radius_m)
    |   movel([0.330796, -0.551267, -2.829943, -1.331179, 1.570796, 1.901592],accel_mss,speed_ms,0,blend_radius_m)
    |   movel([0.333311, -0.545845, -2.830262, -1.336282, 1.570796, 1.904108],accel_mss,speed_ms,0,blend_radius_m)
    |   movel([0.335025, -0.541365, -2.830517, -1.340507, 1.570796, 1.905822],accel_mss,speed_ms,0,blend_radius_m)
    |   movel([0.336222, -0.537186, -2.830749, -1.344454, 1.570796, 1.907018],accel_mss,speed_ms,0,blend_radius_m)
    |   movel([0.336873, -0.533393, -2.830954, -1.348042, 1.570796, 1.907669],accel_mss,speed_ms,0,blend_radius_m)
    |   movel([0.336955, -0.530077, -2.831129, -1.351183, 1.570796, 1.907752],accel_mss,speed_ms,0,blend_radius_m)
    |   movel([0.338790, -0.528590, -2.831206, -1.352593, 1.570796, 1.909587],accel_mss,speed_ms,0,blend_radius_m)
    |   movel([0.340535, -0.527532, -2.831260, -1.353597, 1.570796, 1.911331],accel_mss,speed_ms,0,blend_radius_m)
    |   movel([0.343881, -0.525961, -2.831340, -1.355088, 1.570796, 1.914677],accel_mss,speed_ms,0,blend_radius_m)
    |   movel([0.347442, -0.523990, -2.831440, -1.356959, 1.570796, 1.918238],accel_mss,speed_ms,0,blend_radius_m)
    |   movel([0.349291, -0.522541, -2.831512, -1.358337, 1.570796, 1.920088],accel_mss,speed_ms,0,blend_radius_m)
    |   movel([0.351095, -0.520631, -2.831605, -1.360152, 1.570796, 1.921891],accel_mss,speed_ms,0,blend_radius_m)
    |   movel([0.371911, -0.495429, -2.832725, -1.384235, 1.570796, 1.942707],accel_mss,speed_ms,0,blend_radius_m)
    |   movel([0.372322, -0.492808, -2.832828, -1.386752, 1.570796, 1.943119],accel_mss,speed_ms,0,blend_radius_m)
    |   movel([0.371894, -0.490872, -2.832904, -1.388614, 1.570796, 1.942690],accel_mss,speed_ms,0,blend_radius_m)
    |   movel([0.370646, -0.489723, -2.832948, -1.389718, 1.570796, 1.941442],accel_mss,speed_ms,0,blend_radius_m)
    |   movel([0.368631, -0.489448, -2.832958, -1.389983, 1.570796, 1.939427],accel_mss,speed_ms,0,blend_radius_m)
    |   movel([0.372880, -0.486714, -2.833061, -1.392614, 1.570796, 1.943676],accel_mss,speed_ms,0,blend_radius_m)
    |   movel([0.376752, -0.484875, -2.833128, -1.394385, 1.570796, 1.947549],accel_mss,speed_ms,0,blend_radius_m)
    |   movel([0.380046, -0.484013, -2.833159, -1.395217, 1.570796, 1.950842],accel_mss,speed_ms,0,blend_radius_m)
    |   movel([0.382576, -0.484196, -2.833153, -1.395040, 1.570796, 1.953372],accel_mss,speed_ms,0,blend_radius_m)
    |   speed_ms = 0.005
    |   movel([0.382576, -0.480586, -2.826179, -1.405623, 1.570796, 1.953372],accel_mss,speed_ms,0,blend_radius_m)
    |   speed_ms = 0.040
    |   movel([0.387026, -0.469083, -2.826572, -1.416734, 1.570796, 1.957822],accel_mss,speed_ms,0,blend_radius_m)
    |   speed_ms = 0.005
    |   movel([0.387026, -0.472461, -2.833554, -1.406374, 1.570796, 1.957822],accel_mss,speed_ms,0,blend_radius_m)
    |   speed_ms = 0.025
    |   movel([0.390234, -0.465861, -2.833759, -1.412769, 1.570796, 1.961030],accel_mss,speed_ms,0,blend_radius_m)
    |   movel([0.392915, -0.459713, -2.833937, -1.418739, 1.570796, 1.963711],accel_mss,speed_ms,0,blend_radius_m)
    |   movel([0.395105, -0.453970, -2.834091, -1.424328, 1.570796, 1.965901],accel_mss,speed_ms,0,blend_radius_m)
    |   movel([0.396834, -0.448586, -2.834226, -1.429577, 1.570796, 1.967631],accel_mss,speed_ms,0,blend_radius_m)
    |   movel([0.398138, -0.443507, -2.834344, -1.434538, 1.570796, 1.968935],accel_mss,speed_ms,0,blend_radius_m)
    |   movel([0.399054, -0.438677, -2.834449, -1.439263, 1.570796, 1.969851],accel_mss,speed_ms,0,blend_radius_m)
    |   movel([0.399874, -0.429554, -2.834625, -1.448210, 1.570796, 1.970670],accel_mss,speed_ms,0,blend_radius_m)
    |   movel([0.388878, -0.452327, -2.834133, -1.425928, 1.570796, 1.959675],accel_mss,speed_ms,0,blend_radius_m)
    |   movel([0.389879, -0.449919, -2.834194, -1.428277, 1.570796, 1.960676],accel_mss,speed_ms,0,blend_radius_m)
    |   movel([0.390488, -0.447764, -2.834246, -1.430379, 1.570796, 1.961284],accel_mss,speed_ms,0,blend_radius_m)
    |   movel([0.390661, -0.444174, -2.834329, -1.433885, 1.570796, 1.961457],accel_mss,speed_ms,0,blend_radius_m)
    |   movel([0.389642, -0.441478, -2.834389, -1.436522, 1.570796, 1.960438],accel_mss,speed_ms,0,blend_radius_m)
    |   movel([0.387713, -0.439584, -2.834430, -1.438376, 1.570796, 1.958510],accel_mss,speed_ms,0,blend_radius_m)
    |   movel([0.385147, -0.438385, -2.834455, -1.439549, 1.570796, 1.955943],accel_mss,speed_ms,0,blend_radius_m)
    |   movel([0.382231, -0.437781, -2.834467, -1.440141, 1.570796, 1.953027],accel_mss,speed_ms,0,blend_radius_m)
    |   movel([0.376502, -0.437900, -2.834465, -1.440024, 1.570796, 1.947298],accel_mss,speed_ms,0,blend_radius_m)
    |   movel([0.377900, -0.444257, -2.834327, -1.433804, 1.570796, 1.948696],accel_mss,speed_ms,0,blend_radius_m)
    |   movel([0.377790, -0.448279, -2.834233, -1.429877, 1.570796, 1.948587],accel_mss,speed_ms,0,blend_radius_m)
    |   movel([0.376630, -0.452871, -2.834119, -1.425399, 1.570796, 1.947427],accel_mss,speed_ms,0,blend_radius_m)
    |   movel([0.374047, -0.453905, -2.834093, -1.424391, 1.570796, 1.944843],accel_mss,speed_ms,0,blend_radius_m)
    |   movel([0.371733, -0.454368, -2.834081, -1.423940, 1.570796, 1.942530],accel_mss,speed_ms,0,blend_radius_m)
    |   movel([0.367508, -0.454355, -2.834081, -1.423953, 1.570796, 1.938304],accel_mss,speed_ms,0,blend_radius_m)
    |   movel([0.363181, -0.454342, -2.834081, -1.423965, 1.570796, 1.933977],accel_mss,speed_ms,0,blend_radius_m)
    |   movel([0.360741, -0.454805, -2.834069, -1.423515, 1.570796, 1.931537],accel_mss,speed_ms,0,blend_radius_m)
    |   movel([0.358006, -0.455815, -2.834043, -1.422532, 1.570796, 1.928802],accel_mss,speed_ms,0,blend_radius_m)
    |   movel([0.354695, -0.461853, -2.833876, -1.416660, 1.570796, 1.925492],accel_mss,speed_ms,0,blend_radius_m)
    |   movel([0.352388, -0.467412, -2.833712, -1.411265, 1.570796, 1.923184],accel_mss,speed_ms,0,blend_radius_m)
    |   movel([0.348526, -0.469341, -2.833653, -1.409396, 1.570796, 1.919323],accel_mss,speed_ms,0,blend_radius_m)
    |   movel([0.345063, -0.470496, -2.833616, -1.408277, 1.570796, 1.915860],accel_mss,speed_ms,0,blend_radius_m)
    |   movel([0.342063, -0.470856, -2.833605, -1.407928, 1.570796, 1.912860],accel_mss,speed_ms,0,blend_radius_m)
    |   movel([0.339611, -0.470408, -2.833619, -1.408361, 1.570796, 1.910407],accel_mss,speed_ms,0,blend_radius_m)
    |   movel([0.339108, -0.471071, -2.833598, -1.407720, 1.570796, 1.909904],accel_mss,speed_ms,0,blend_radius_m)
    |   movel([0.334776, -0.478623, -2.833349, -1.400417, 1.570796, 1.905572],accel_mss,speed_ms,0,blend_radius_m)
    |   movel([0.329791, -0.487877, -2.833017, -1.391494, 1.570796, 1.900587],accel_mss,speed_ms,0,blend_radius_m)
    |   movel([0.327876, -0.492145, -2.832854, -1.387389, 1.570796, 1.898672],accel_mss,speed_ms,0,blend_radius_m)
    |   movel([0.326434, -0.495936, -2.832704, -1.383748, 1.570796, 1.897230],accel_mss,speed_ms,0,blend_radius_m)
    |   movel([0.324271, -0.503333, -2.832397, -1.376659, 1.570796, 1.895068],accel_mss,speed_ms,0,blend_radius_m)
    |   movel([0.316314, -0.500074, -2.832535, -1.379780, 1.570796, 1.887111],accel_mss,speed_ms,0,blend_radius_m)
    |   movel([0.314190, -0.504589, -2.832344, -1.375457, 1.570796, 1.884986],accel_mss,speed_ms,0,blend_radius_m)
    |   movel([0.312390, -0.508971, -2.832151, -1.371267, 1.570796, 1.883187],accel_mss,speed_ms,0,blend_radius_m)
    |   movel([0.309655, -0.517307, -2.831766, -1.363316, 1.570796, 1.880451],accel_mss,speed_ms,0,blend_radius_m)
    |   movel([0.307967, -0.524916, -2.831393, -1.356080, 1.570796, 1.878764],accel_mss,speed_ms,0,blend_radius_m)
    |   movel([0.306909, -0.533722, -2.830936, -1.347730, 1.570796, 1.877705],accel_mss,speed_ms,0,blend_radius_m)
    |   movel([0.306515, -0.534911, -2.830872, -1.346606, 1.570796, 1.877311],accel_mss,speed_ms,0,blend_radius_m)
    |   movel([0.305827, -0.536216, -2.830802, -1.345371, 1.570796, 1.876623],accel_mss,speed_ms,0,blend_radius_m)
    |   movel([0.304478, -0.537962, -2.830706, -1.343721, 1.570796, 1.875274],accel_mss,speed_ms,0,blend_radius_m)
    |   movel([0.294561, -0.547901, -2.830142, -1.334346, 1.570796, 1.865358],accel_mss,speed_ms,0,blend_radius_m)
    |   movel([0.289552, -0.552304, -2.829881, -1.330203, 1.570796, 1.860349],accel_mss,speed_ms,0,blend_radius_m)
    |   movel([0.287733, -0.553514, -2.829808, -1.329067, 1.570796, 1.858529],accel_mss,speed_ms,0,blend_radius_m)
    |   movel([0.286703, -0.553666, -2.829799, -1.328924, 1.570796, 1.857500],accel_mss,speed_ms,0,blend_radius_m)
    |   movel([0.290558, -0.555934, -2.829661, -1.326794, 1.570796, 1.861354],accel_mss,speed_ms,0,blend_radius_m)
    |   movel([0.292858, -0.556555, -2.829622, -1.326212, 1.570796, 1.863654],accel_mss,speed_ms,0,blend_radius_m)
    |   movel([0.295384, -0.556840, -2.829605, -1.325945, 1.570796, 1.866180],accel_mss,speed_ms,0,blend_radius_m)
    |   movel([0.286906, -0.567939, -2.828897, -1.315553, 1.570796, 1.857702],accel_mss,speed_ms,0,blend_radius_m)
    |   movel([0.278033, -0.580104, -2.828068, -1.304217, 1.570796, 1.848829],accel_mss,speed_ms,0,blend_radius_m)
    |   movel([0.273863, -0.586218, -2.827631, -1.298540, 1.570796, 1.844659],accel_mss,speed_ms,0,blend_radius_m)
    |   movel([0.270079, -0.592154, -2.827193, -1.293042, 1.570796, 1.840875],accel_mss,speed_ms,0,blend_radius_m)
    |   movel([0.266838, -0.597781, -2.826766, -1.287842, 1.570796, 1.837635],accel_mss,speed_ms,0,blend_radius_m)
    |   movel([0.264289, -0.602955, -2.826363, -1.283071, 1.570796, 1.835085],accel_mss,speed_ms,0,blend_radius_m)
    |   movel([0.268149, -0.598810, -2.826687, -1.286892, 1.570796, 1.838945],accel_mss,speed_ms,0,blend_radius_m)
    |   movel([0.272090, -0.594973, -2.826981, -1.290435, 1.570796, 1.842886],accel_mss,speed_ms,0,blend_radius_m)
    |   movel([0.276063, -0.591528, -2.827240, -1.293621, 1.570796, 1.846859],accel_mss,speed_ms,0,blend_radius_m)
    |   movel([0.280040, -0.588544, -2.827461, -1.296384, 1.570796, 1.850836],accel_mss,speed_ms,0,blend_radius_m)
    |   movel([0.277321, -0.591868, -2.827215, -1.293306, 1.570796, 1.848118],accel_mss,speed_ms,0,blend_radius_m)
    |   movel([0.272341, -0.598742, -2.826692, -1.286955, 1.570796, 1.843137],accel_mss,speed_ms,0,blend_radius_m)
    |   movel([0.270112, -0.602236, -2.826419, -1.283734, 1.570796, 1.840909],accel_mss,speed_ms,0,blend_radius_m)
    |   movel([0.266283, -0.609142, -2.825867, -1.277380, 1.570796, 1.837079],accel_mss,speed_ms,0,blend_radius_m)
    |   movel([0.264712, -0.612503, -2.825591, -1.274295, 1.570796, 1.835509],accel_mss,speed_ms,0,blend_radius_m)
    |   movel([0.263401, -0.615752, -2.825320, -1.271316, 1.570796, 1.834197],accel_mss,speed_ms,0,blend_radius_m)
    |   speed_ms = 0.005
    |   movel([0.263401, -0.609750, -2.818510, -1.284129, 1.570796, 1.834197],accel_mss,speed_ms,0,blend_radius_m)
    |   speed_ms = 0.040
    |   movel([0.276538, -0.610567, -2.818442, -1.283380, 1.570796, 1.847334],accel_mss,speed_ms,0,blend_radius_m)
    |   speed_ms = 0.005
    |   movel([0.276538, -0.616584, -2.825250, -1.270555, 1.570796, 1.847334],accel_mss,speed_ms,0,blend_radius_m)
    |   speed_ms = 0.025
    |   movel([0.277545, -0.612524, -2.825589, -1.274276, 1.570796, 1.848342],accel_mss,speed_ms,0,blend_radius_m)
    |   movel([0.278896, -0.608213, -2.825942, -1.278234, 1.570796, 1.849693],accel_mss,speed_ms,0,blend_radius_m)
    |   movel([0.280584, -0.603691, -2.826304, -1.282393, 1.570796, 1.851380],accel_mss,speed_ms,0,blend_radius_m)
    |   movel([0.282599, -0.599005, -2.826672, -1.286713, 1.570796, 1.853396],accel_mss,speed_ms,0,blend_radius_m)
    |   movel([0.284943, -0.594184, -2.827041, -1.291164, 1.570796, 1.855739],accel_mss,speed_ms,0,blend_radius_m)
    |   movel([0.287601, -0.589277, -2.827407, -1.295705, 1.570796, 1.858397],accel_mss,speed_ms,0,blend_radius_m)
    |   movel([0.290566, -0.584319, -2.827769, -1.300302, 1.570796, 1.861362],accel_mss,speed_ms,0,blend_radius_m)
    |   movel([0.293832, -0.579358, -2.828121, -1.304910, 1.570796, 1.864628],accel_mss,speed_ms,0,blend_radius_m)
    |   movel([0.304616, -0.563878, -2.829161, -1.319350, 1.570796, 1.875413],accel_mss,speed_ms,0,blend_radius_m)
    |   movel([0.306870, -0.560261, -2.829391, -1.322737, 1.570796, 1.877667],accel_mss,speed_ms,0,blend_radius_m)
    |   movel([0.308921, -0.556569, -2.829621, -1.326199, 1.570796, 1.879718],accel_mss,speed_ms,0,blend_radius_m)
    |   movel([0.310757, -0.552722, -2.829856, -1.329811, 1.570796, 1.881553],accel_mss,speed_ms,0,blend_radius_m)
    |   movel([0.312371, -0.548619, -2.830100, -1.333669, 1.570796, 1.883168],accel_mss,speed_ms,0,blend_radius_m)
    |   movel([0.315959, -0.537307, -2.830742, -1.344340, 1.570796, 1.886755],accel_mss,speed_ms,0,blend_radius_m)
    |   movel([0.318021, -0.531504, -2.831054, -1.349831, 1.570796, 1.888818],accel_mss,speed_ms,0,blend_radius_m)
    |   movel([0.320838, -0.525314, -2.831373, -1.355702, 1.570796, 1.891635],accel_mss,speed_ms,0,blend_radius_m)
    |   movel([0.323030, -0.521386, -2.831569, -1.359434, 1.570796, 1.893826],accel_mss,speed_ms,0,blend_radius_m)
    |   movel([0.325522, -0.517422, -2.831760, -1.363206, 1.570796, 1.896318],accel_mss,speed_ms,0,blend_radius_m)
    |   movel([0.331230, -0.509449, -2.832129, -1.370811, 1.570796, 1.902027],accel_mss,speed_ms,0,blend_radius_m)
    |   movel([0.337587, -0.501492, -2.832476, -1.378421, 1.570796, 1.908384],accel_mss,speed_ms,0,blend_radius_m)
    |   movel([0.344229, -0.493653, -2.832795, -1.385941, 1.570796, 1.915025],accel_mss,speed_ms,0,blend_radius_m)
    |   movel([0.350788, -0.486151, -2.833081, -1.393157, 1.570796, 1.921584],accel_mss,speed_ms,0,blend_radius_m)
    |   movel([0.357574, -0.478938, -2.833338, -1.400113, 1.570796, 1.928371],accel_mss,speed_ms,0,blend_radius_m)
    |   movel([0.360967, -0.475666, -2.833449, -1.403274, 1.570796, 1.931763],accel_mss,speed_ms,0,blend_radius_m)
    |   movel([0.364324, -0.472726, -2.833545, -1.406118, 1.570796, 1.935120],accel_mss,speed_ms,0,blend_radius_m)
    |   movel([0.367586, -0.470230, -2.833625, -1.408534, 1.570796, 1.938382],accel_mss,speed_ms,0,blend_radius_m)
    |   movel([0.370742, -0.468246, -2.833686, -1.410457, 1.570796, 1.941538],accel_mss,speed_ms,0,blend_radius_m)
    |   speed_ms = 0.005
    |   movel([0.370742, -0.464951, -2.826701, -1.420736, 1.570796, 1.941538],accel_mss,speed_ms,0,blend_radius_m)
    |   speed_ms = 0.040
    |   movel([0.373720, -0.466431, -2.826656, -1.419302, 1.570796, 1.944517],accel_mss,speed_ms,0,blend_radius_m)
    |   speed_ms = 0.005
    |   movel([0.373720, -0.469756, -2.833640, -1.408994, 1.570796, 1.944517],accel_mss,speed_ms,0,blend_radius_m)
    |   speed_ms = 0.025
    |   movel([0.374696, -0.470074, -2.833630, -1.408685, 1.570796, 1.945493],accel_mss,speed_ms,0,blend_radius_m)
    |   movel([0.375927, -0.470855, -2.833605, -1.407929, 1.570796, 1.946724],accel_mss,speed_ms,0,blend_radius_m)
    |   movel([0.377343, -0.474200, -2.833497, -1.404692, 1.570796, 1.948140],accel_mss,speed_ms,0,blend_radius_m)
    |   movel([0.377538, -0.476423, -2.833424, -1.402543, 1.570796, 1.948335],accel_mss,speed_ms,0,blend_radius_m)
    |   movel([0.377239, -0.477787, -2.833378, -1.401224, 1.570796, 1.948036],accel_mss,speed_ms,0,blend_radius_m)
    |   movel([0.376871, -0.478236, -2.833362, -1.400790, 1.570796, 1.947667],accel_mss,speed_ms,0,blend_radius_m)
    |   movel([0.376302, -0.478425, -2.833356, -1.400608, 1.570796, 1.947098],accel_mss,speed_ms,0,blend_radius_m)
    |   movel([0.371035, -0.478308, -2.833360, -1.400721, 1.570796, 1.941831],accel_mss,speed_ms,0,blend_radius_m)
    |   movel([0.367919, -0.479015, -2.833336, -1.400038, 1.570796, 1.938716],accel_mss,speed_ms,0,blend_radius_m)
    |   movel([0.366130, -0.479864, -2.833306, -1.399219, 1.570796, 1.936927],accel_mss,speed_ms,0,blend_radius_m)
    |   movel([0.364146, -0.481140, -2.833262, -1.397987, 1.570796, 1.934942],accel_mss,speed_ms,0,blend_radius_m)
    |   movel([0.361793, -0.483080, -2.833193, -1.396116, 1.570796, 1.932589],accel_mss,speed_ms,0,blend_radius_m)
    |   movel([0.359416, -0.485331, -2.833111, -1.393947, 1.570796, 1.930212],accel_mss,speed_ms,0,blend_radius_m)
    |   movel([0.353627, -0.491295, -2.832887, -1.388207, 1.570796, 1.924423],accel_mss,speed_ms,0,blend_radius_m)
    |   movel([0.347921, -0.497688, -2.832633, -1.382067, 1.570796, 1.918717],accel_mss,speed_ms,0,blend_radius_m)
    |   movel([0.342472, -0.504308, -2.832356, -1.375725, 1.570796, 1.913268],accel_mss,speed_ms,0,blend_radius_m)
    |   movel([0.337468, -0.510927, -2.832063, -1.369399, 1.570796, 1.908264],accel_mss,speed_ms,0,blend_radius_m)
    |   movel([0.339354, -0.515490, -2.831852, -1.365047, 1.570796, 1.910150],accel_mss,speed_ms,0,blend_radius_m)
    |   movel([0.340331, -0.520992, -2.831588, -1.359809, 1.570796, 1.911128],accel_mss,speed_ms,0,blend_radius_m)
    |   movel([0.338418, -0.520811, -2.831597, -1.359981, 1.570796, 1.909214],accel_mss,speed_ms,0,blend_radius_m)
    |   movel([0.336083, -0.521316, -2.831572, -1.359501, 1.570796, 1.906879],accel_mss,speed_ms,0,blend_radius_m)
    |   movel([0.333398, -0.522499, -2.831514, -1.358376, 1.570796, 1.904194],accel_mss,speed_ms,0,blend_radius_m)
    |   movel([0.330464, -0.524312, -2.831423, -1.356654, 1.570796, 1.901261],accel_mss,speed_ms,0,blend_radius_m)
    |   movel([0.329011, -0.525642, -2.831356, -1.355391, 1.570796, 1.899807],accel_mss,speed_ms,0,blend_radius_m)
    |   movel([0.328274, -0.527111, -2.831282, -1.353997, 1.570796, 1.899070],accel_mss,speed_ms,0,blend_radius_m)
    |   movel([0.323122, -0.541773, -2.830494, -1.340122, 1.570796, 1.893918],accel_mss,speed_ms,0,blend_radius_m)
    |   movel([0.320044, -0.549431, -2.830052, -1.332906, 1.570796, 1.890841],accel_mss,speed_ms,0,blend_radius_m)
    |   movel([0.316496, -0.557382, -2.829571, -1.325435, 1.570796, 1.887292],accel_mss,speed_ms,0,blend_radius_m)
    |   movel([0.312512, -0.565433, -2.829060, -1.317896, 1.570796, 1.883309],accel_mss,speed_ms,0,blend_radius_m)
    |   movel([0.308113, -0.573409, -2.828531, -1.310449, 1.570796, 1.878909],accel_mss,speed_ms,0,blend_radius_m)
    |   movel([0.298999, -0.589375, -2.827400, -1.295614, 1.570796, 1.869795],accel_mss,speed_ms,0,blend_radius_m)
    |   movel([0.295170, -0.597042, -2.826823, -1.288524, 1.570796, 1.865966],accel_mss,speed_ms,0,blend_radius_m)
    |   movel([0.292205, -0.604448, -2.826244, -1.281697, 1.570796, 1.863001],accel_mss,speed_ms,0,blend_radius_m)
    |   speed_ms = 0.005
    |   movel([0.292205, -0.598635, -2.819415, -1.294339, 1.570796, 1.863001],accel_mss,speed_ms,0,blend_radius_m)
    |   speed_ms = 0.040
    |   movel([0.321661, -0.576562, -2.821071, -1.314756, 1.570796, 1.892458],accel_mss,speed_ms,0,blend_radius_m)
    |   speed_ms = 0.005
    |   movel([0.321661, -0.581990, -2.827935, -1.302464, 1.570796, 1.892458],accel_mss,speed_ms,0,blend_radius_m)
    |   speed_ms = 0.025
    |   movel([0.319197, -0.588063, -2.827497, -1.296829, 1.570796, 1.889993],accel_mss,speed_ms,0,blend_radius_m)
    |   movel([0.315954, -0.594401, -2.827024, -1.290963, 1.570796, 1.886750],accel_mss,speed_ms,0,blend_radius_m)
    |   movel([0.312056, -0.600786, -2.826533, -1.285070, 1.570796, 1.882852],accel_mss,speed_ms,0,blend_radius_m)
    |   movel([0.307630, -0.607016, -2.826039, -1.279334, 1.570796, 1.878426],accel_mss,speed_ms,0,blend_radius_m)
    |   speed_ms = 0.005
    |   movel([0.307630, -0.601159, -2.819214, -1.292016, 1.570796, 1.878426],accel_mss,speed_ms,0,blend_radius_m)
    |   speed_ms = 0.040
    |   movel([0.302674, -0.597103, -2.819536, -1.295750, 1.570796, 1.873470],accel_mss,speed_ms,0,blend_radius_m)
    |   speed_ms = 0.005
    |   movel([0.302674, -0.602890, -2.826368, -1.283131, 1.570796, 1.873470],accel_mss,speed_ms,0,blend_radius_m)
    |   speed_ms = 0.025
    |   movel([0.280331, -0.642157, -2.822967, -1.247265, 1.570796, 1.851128],accel_mss,speed_ms,0,blend_radius_m)
    |   movel([0.279220, -0.644558, -2.822739, -1.245092, 1.570796, 1.850016],accel_mss,speed_ms,0,blend_radius_m)
    |   movel([0.279226, -0.646698, -2.822534, -1.243157, 1.570796, 1.850023],accel_mss,speed_ms,0,blend_radius_m)
    |   movel([0.279227, -0.649463, -2.822267, -1.240659, 1.570796, 1.850024],accel_mss,speed_ms,0,blend_radius_m)
    |   movel([0.278517, -0.652766, -2.821943, -1.237680, 1.570796, 1.849314],accel_mss,speed_ms,0,blend_radius_m)
    |   speed_ms = 0.005
    |   movel([0.278517, -0.646169, -2.815201, -1.251019, 1.570796, 1.849314],accel_mss,speed_ms,0,blend_radius_m)
    |   speed_ms = 0.040
    |   movel([0.311735, -0.616669, -2.817922, -1.277798, 1.570796, 1.882531],accel_mss,speed_ms,0,blend_radius_m)
    |   speed_ms = 0.005
    |   movel([0.311735, -0.622788, -2.824720, -1.264881, 1.570796, 1.882531],accel_mss,speed_ms,0,blend_radius_m)
    |   speed_ms = 0.025
    |   movel([0.312655, -0.619139, -2.825034, -1.268216, 1.570796, 1.883451],accel_mss,speed_ms,0,blend_radius_m)
    |   movel([0.314010, -0.615224, -2.825364, -1.271800, 1.570796, 1.884807],accel_mss,speed_ms,0,blend_radius_m)
    |   movel([0.315778, -0.611109, -2.825706, -1.275574, 1.570796, 1.886574],accel_mss,speed_ms,0,blend_radius_m)
    |   movel([0.317946, -0.606841, -2.826053, -1.279496, 1.570796, 1.888742],accel_mss,speed_ms,0,blend_radius_m)
    |   movel([0.319684, -0.603833, -2.826293, -1.282263, 1.570796, 1.890481],accel_mss,speed_ms,0,blend_radius_m)
    |   movel([0.321646, -0.600819, -2.826530, -1.285039, 1.570796, 1.892442],accel_mss,speed_ms,0,blend_radius_m)
    |   movel([0.323814, -0.597921, -2.826755, -1.287713, 1.570796, 1.894611],accel_mss,speed_ms,0,blend_radius_m)
    |   movel([0.326196, -0.595227, -2.826962, -1.290200, 1.570796, 1.896993],accel_mss,speed_ms,0,blend_radius_m)
    |   movel([0.328279, -0.593334, -2.827105, -1.291950, 1.570796, 1.899076],accel_mss,speed_ms,0,blend_radius_m)
    |   movel([0.330485, -0.591760, -2.827223, -1.293406, 1.570796, 1.901281],accel_mss,speed_ms,0,blend_radius_m)
    |   movel([0.332750, -0.590469, -2.827319, -1.294601, 1.570796, 1.903546],accel_mss,speed_ms,0,blend_radius_m)
    |   movel([0.335028, -0.589420, -2.827397, -1.295572, 1.570796, 1.905824],accel_mss,speed_ms,0,blend_radius_m)
    |   movel([0.339388, -0.587888, -2.827509, -1.296991, 1.570796, 1.910184],accel_mss,speed_ms,0,blend_radius_m)
    |   movel([0.343127, -0.586855, -2.827585, -1.297949, 1.570796, 1.913924],accel_mss,speed_ms,0,blend_radius_m)
    |   movel([0.340461, -0.587851, -2.827512, -1.297026, 1.570796, 1.911258],accel_mss,speed_ms,0,blend_radius_m)
    |   movel([0.337596, -0.589473, -2.827393, -1.295523, 1.570796, 1.908393],accel_mss,speed_ms,0,blend_radius_m)
    |   movel([0.334582, -0.591759, -2.827223, -1.293407, 1.570796, 1.905378],accel_mss,speed_ms,0,blend_radius_m)
    |   movel([0.331459, -0.594762, -2.826997, -1.290630, 1.570796, 1.902255],accel_mss,speed_ms,0,blend_radius_m)
    |   movel([0.328877, -0.597792, -2.826765, -1.287831, 1.570796, 1.899674],accel_mss,speed_ms,0,blend_radius_m)
    |   movel([0.326509, -0.601012, -2.826515, -1.284862, 1.570796, 1.897306],accel_mss,speed_ms,0,blend_radius_m)
    |   movel([0.324448, -0.604144, -2.826268, -1.281977, 1.570796, 1.895244],accel_mss,speed_ms,0,blend_radius_m)
    |   movel([0.322628, -0.607269, -2.826018, -1.279101, 1.570796, 1.893424],accel_mss,speed_ms,0,blend_radius_m)
    |   movel([0.319681, -0.613406, -2.825516, -1.273467, 1.570796, 1.890478],accel_mss,speed_ms,0,blend_radius_m)
    |   movel([0.317617, -0.619209, -2.825028, -1.268152, 1.570796, 1.888413],accel_mss,speed_ms,0,blend_radius_m)
    |   movel([0.316306, -0.624919, -2.824534, -1.262935, 1.570796, 1.887102],accel_mss,speed_ms,0,blend_radius_m)
    |   speed_ms = 0.005
    |   movel([0.316306, -0.618766, -2.817740, -1.275883, 1.570796, 1.887102],accel_mss,speed_ms,0,blend_radius_m)
    |   speed_ms = 0.040
    |   movel([0.326073, -0.603824, -2.818999, -1.289566, 1.570796, 1.896869],accel_mss,speed_ms,0,blend_radius_m)
    |   speed_ms = 0.005
    |   movel([0.326073, -0.609726, -2.825819, -1.276844, 1.570796, 1.896869],accel_mss,speed_ms,0,blend_radius_m)
    |   speed_ms = 0.025
    |   movel([0.325521, -0.610698, -2.825739, -1.275952, 1.570796, 1.896317],accel_mss,speed_ms,0,blend_radius_m)
    |   movel([0.324673, -0.611352, -2.825686, -1.275351, 1.570796, 1.895469],accel_mss,speed_ms,0,blend_radius_m)
    |   movel([0.324243, -0.611132, -2.825704, -1.275553, 1.570796, 1.895039],accel_mss,speed_ms,0,blend_radius_m)
    |   movel([0.324311, -0.610338, -2.825769, -1.276282, 1.570796, 1.895107],accel_mss,speed_ms,0,blend_radius_m)
    |   movel([0.325465, -0.608241, -2.825940, -1.278208, 1.570796, 1.896261],accel_mss,speed_ms,0,blend_radius_m)
    |   movel([0.326191, -0.607339, -2.826013, -1.279037, 1.570796, 1.896987],accel_mss,speed_ms,0,blend_radius_m)
    |   movel([0.326922, -0.606987, -2.826041, -1.279361, 1.570796, 1.897719],accel_mss,speed_ms,0,blend_radius_m)
    |   movel([0.327219, -0.607401, -2.826008, -1.278981, 1.570796, 1.898015],accel_mss,speed_ms,0,blend_radius_m)
    |   movel([0.326594, -0.609267, -2.825856, -1.277266, 1.570796, 1.897391],accel_mss,speed_ms,0,blend_radius_m)
    |   speed_ms = 0.005
    |   movel([0.326594, -0.603372, -2.819035, -1.289981, 1.570796, 1.897391],accel_mss,speed_ms,0,blend_radius_m)
    |   speed_ms = 0.040
    |   movel([0.322157, -0.625491, -2.817145, -1.269753, 1.570796, 1.892954],accel_mss,speed_ms,0,blend_radius_m)
    |   speed_ms = 0.005
    |   movel([0.322157, -0.631755, -2.823927, -1.256707, 1.570796, 1.892954],accel_mss,speed_ms,0,blend_radius_m)
    |   speed_ms = 0.025
    |   movel([0.325186, -0.627820, -2.824279, -1.260290, 1.570796, 1.895982],accel_mss,speed_ms,0,blend_radius_m)
    |   movel([0.327817, -0.623858, -2.824627, -1.263904, 1.570796, 1.898613],accel_mss,speed_ms,0,blend_radius_m)
    |   movel([0.333129, -0.615844, -2.825313, -1.271233, 1.570796, 1.903926],accel_mss,speed_ms,0,blend_radius_m)
    |   movel([0.337484, -0.610310, -2.825771, -1.276308, 1.570796, 1.908280],accel_mss,speed_ms,0,blend_radius_m)
    |   movel([0.351880, -0.593791, -2.827070, -1.291527, 1.570796, 1.922677],accel_mss,speed_ms,0,blend_radius_m)
    |   movel([0.354699, -0.590147, -2.827343, -1.294899, 1.570796, 1.925495],accel_mss,speed_ms,0,blend_radius_m)
    |   movel([0.355695, -0.588389, -2.827473, -1.296527, 1.570796, 1.926491],accel_mss,speed_ms,0,blend_radius_m)
    |   movel([0.356078, -0.586934, -2.827579, -1.297876, 1.570796, 1.926874],accel_mss,speed_ms,0,blend_radius_m)
    |   movel([0.355513, -0.586026, -2.827645, -1.298718, 1.570796, 1.926310],accel_mss,speed_ms,0,blend_radius_m)
    |   movel([0.354294, -0.585914, -2.827653, -1.298822, 1.570796, 1.925091],accel_mss,speed_ms,0,blend_radius_m)
    |   movel([0.352221, -0.586235, -2.827630, -1.298524, 1.570796, 1.923017],accel_mss,speed_ms,0,blend_radius_m)
    |   movel([0.350044, -0.587141, -2.827564, -1.297684, 1.570796, 1.920840],accel_mss,speed_ms,0,blend_radius_m)
    |   movel([0.347607, -0.588746, -2.827446, -1.296197, 1.570796, 1.918404],accel_mss,speed_ms,0,blend_radius_m)
    |   movel([0.344764, -0.591149, -2.827268, -1.293971, 1.570796, 1.915560],accel_mss,speed_ms,0,blend_radius_m)
    |   movel([0.341697, -0.594225, -2.827038, -1.291127, 1.570796, 1.912493],accel_mss,speed_ms,0,blend_radius_m)
    |   movel([0.338653, -0.597747, -2.826769, -1.287873, 1.570796, 1.909450],accel_mss,speed_ms,0,blend_radius_m)
    |   movel([0.335674, -0.601577, -2.826471, -1.284341, 1.570796, 1.906470],accel_mss,speed_ms,0,blend_radius_m)
    |   movel([0.332788, -0.605606, -2.826152, -1.280631, 1.570796, 1.903584],accel_mss,speed_ms,0,blend_radius_m)
    |   movel([0.327453, -0.613724, -2.825490, -1.273175, 1.570796, 1.898250],accel_mss,speed_ms,0,blend_radius_m)
    |   movel([0.322905, -0.621134, -2.824863, -1.266392, 1.570796, 1.893702],accel_mss,speed_ms,0,blend_radius_m)
    |   movel([0.314910, -0.634729, -2.823657, -1.254003, 1.570796, 1.885707],accel_mss,speed_ms,0,blend_radius_m)
    |   movel([0.312085, -0.639189, -2.823245, -1.249955, 1.570796, 1.882881],accel_mss,speed_ms,0,blend_radius_m)
    |   movel([0.308996, -0.643601, -2.822830, -1.245958, 1.570796, 1.879792],accel_mss,speed_ms,0,blend_radius_m)
    |   movel([0.305647, -0.647811, -2.822427, -1.242151, 1.570796, 1.876444],accel_mss,speed_ms,0,blend_radius_m)
    |   movel([0.302132, -0.651587, -2.822059, -1.238743, 1.570796, 1.872929],accel_mss,speed_ms,0,blend_radius_m)
    |   movel([0.298538, -0.654705, -2.821751, -1.235933, 1.570796, 1.869334],accel_mss,speed_ms,0,blend_radius_m)
    |   movel([0.301125, -0.653447, -2.821876, -1.237066, 1.570796, 1.871922],accel_mss,speed_ms,0,blend_radius_m)
    |   movel([0.303822, -0.651857, -2.822033, -1.238500, 1.570796, 1.874618],accel_mss,speed_ms,0,blend_radius_m)
    |   movel([0.306605, -0.649941, -2.822220, -1.240228, 1.570796, 1.877401],accel_mss,speed_ms,0,blend_radius_m)
    |   movel([0.309429, -0.647735, -2.822434, -1.242220, 1.570796, 1.880225],accel_mss,speed_ms,0,blend_radius_m)
    |   movel([0.308725, -0.651065, -2.822110, -1.239214, 1.570796, 1.879521],accel_mss,speed_ms,0,blend_radius_m)
    |   movel([0.307539, -0.654679, -2.821754, -1.235956, 1.570796, 1.878336],accel_mss,speed_ms,0,blend_radius_m)
    |   movel([0.305912, -0.658479, -2.821373, -1.232537, 1.570796, 1.876709],accel_mss,speed_ms,0,blend_radius_m)
    |   movel([0.303882, -0.662376, -2.820976, -1.229037, 1.570796, 1.874679],accel_mss,speed_ms,0,blend_radius_m)
    |   movel([0.307225, -0.658202, -2.821401, -1.232786, 1.570796, 1.878021],accel_mss,speed_ms,0,blend_radius_m)
    |   movel([0.310276, -0.653887, -2.821832, -1.236669, 1.570796, 1.881072],accel_mss,speed_ms,0,blend_radius_m)
    |   movel([0.313052, -0.649464, -2.822267, -1.240658, 1.570796, 1.883848],accel_mss,speed_ms,0,blend_radius_m)
    |   movel([0.315584, -0.644965, -2.822700, -1.244723, 1.570796, 1.886380],accel_mss,speed_ms,0,blend_radius_m)
    |   movel([0.315215, -0.647145, -2.822491, -1.242753, 1.570796, 1.886011],accel_mss,speed_ms,0,blend_radius_m)
    |   movel([0.314349, -0.649807, -2.822233, -1.240349, 1.570796, 1.885146],accel_mss,speed_ms,0,blend_radius_m)
    |   movel([0.308893, -0.662415, -2.820972, -1.229002, 1.570796, 1.879689],accel_mss,speed_ms,0,blend_radius_m)
    |   movel([0.307770, -0.665386, -2.820665, -1.226338, 1.570796, 1.878567],accel_mss,speed_ms,0,blend_radius_m)
    |   movel([0.307040, -0.668007, -2.820392, -1.223991, 1.570796, 1.877836],accel_mss,speed_ms,0,blend_radius_m)
    |   movel([0.309310, -0.663557, -2.820855, -1.227977, 1.570796, 1.880106],accel_mss,speed_ms,0,blend_radius_m)
    |   movel([0.311739, -0.659342, -2.821285, -1.231761, 1.570796, 1.882535],accel_mss,speed_ms,0,blend_radius_m)
    |   movel([0.316962, -0.651340, -2.822083, -1.238966, 1.570796, 1.887758],accel_mss,speed_ms,0,blend_radius_m)
    |   movel([0.322501, -0.643385, -2.822851, -1.246153, 1.570796, 1.893297],accel_mss,speed_ms,0,blend_radius_m)
    |   movel([0.328174, -0.634828, -2.823648, -1.253913, 1.570796, 1.898970],accel_mss,speed_ms,0,blend_radius_m)
    |   movel([0.331292, -0.629470, -2.824132, -1.258787, 1.570796, 1.902088],accel_mss,speed_ms,0,blend_radius_m)
    |   movel([0.333276, -0.626462, -2.824399, -1.261528, 1.570796, 1.904072],accel_mss,speed_ms,0,blend_radius_m)
    |   movel([0.334199, -0.625337, -2.824498, -1.262554, 1.570796, 1.904995],accel_mss,speed_ms,0,blend_radius_m)
    |   movel([0.335018, -0.624631, -2.824560, -1.263199, 1.570796, 1.905814],accel_mss,speed_ms,0,blend_radius_m)
    |   movel([0.335671, -0.624422, -2.824578, -1.263389, 1.570796, 1.906468],accel_mss,speed_ms,0,blend_radius_m)
    |   movel([0.336148, -0.624639, -2.824559, -1.263191, 1.570796, 1.906944],accel_mss,speed_ms,0,blend_radius_m)
    |   movel([0.336625, -0.625970, -2.824442, -1.261977, 1.570796, 1.907421],accel_mss,speed_ms,0,blend_radius_m)
    |   movel([0.336513, -0.627920, -2.824270, -1.260199, 1.570796, 1.907310],accel_mss,speed_ms,0,blend_radius_m)
    |   movel([0.335878, -0.629782, -2.824104, -1.258503, 1.570796, 1.906674],accel_mss,speed_ms,0,blend_radius_m)
    |   movel([0.339381, -0.623014, -2.824700, -1.264674, 1.570796, 1.910177],accel_mss,speed_ms,0,blend_radius_m)
    |   movel([0.342378, -0.616345, -2.825270, -1.270774, 1.570796, 1.913174],accel_mss,speed_ms,0,blend_radius_m)
    |   movel([0.344828, -0.609878, -2.825807, -1.276705, 1.570796, 1.915625],accel_mss,speed_ms,0,blend_radius_m)
    |   movel([0.346680, -0.603710, -2.826303, -1.282376, 1.570796, 1.917476],accel_mss,speed_ms,0,blend_radius_m)
    |   speed_ms = 0.005
    |   movel([0.346680, -0.597909, -2.819473, -1.295007, 1.570796, 1.917476],accel_mss,speed_ms,0,blend_radius_m)
    |   speed_ms = 0.040
    |   movel([0.351511, -0.598011, -2.819465, -1.294914, 1.570796, 1.922307],accel_mss,speed_ms,0,blend_radius_m)
    |   speed_ms = 0.005
    |   movel([0.351511, -0.603814, -2.826295, -1.282281, 1.570796, 1.922307],accel_mss,speed_ms,0,blend_radius_m)
    |   speed_ms = 0.025
    |   movel([0.354434, -0.603525, -2.826317, -1.282547, 1.570796, 1.925230],accel_mss,speed_ms,0,blend_radius_m)
    |   movel([0.355414, -0.604029, -2.826278, -1.282083, 1.570796, 1.926210],accel_mss,speed_ms,0,blend_radius_m)
    |   movel([0.355769, -0.605246, -2.826181, -1.280962, 1.570796, 1.926566],accel_mss,speed_ms,0,blend_radius_m)
    |   movel([0.355477, -0.606833, -2.826053, -1.279503, 1.570796, 1.926273],accel_mss,speed_ms,0,blend_radius_m)
    |   movel([0.345300, -0.636031, -2.823538, -1.252821, 1.570796, 1.916096],accel_mss,speed_ms,0,blend_radius_m)
    |   movel([0.344489, -0.638133, -2.823344, -1.250912, 1.570796, 1.915285],accel_mss,speed_ms,0,blend_radius_m)
    |   movel([0.343421, -0.640318, -2.823140, -1.248931, 1.570796, 1.914218],accel_mss,speed_ms,0,blend_radius_m)
    |   movel([0.342083, -0.642327, -2.822951, -1.247111, 1.570796, 1.912880],accel_mss,speed_ms,0,blend_radius_m)
    |   movel([0.340481, -0.643889, -2.822803, -1.245697, 1.570796, 1.911277],accel_mss,speed_ms,0,blend_radius_m)
    |   movel([0.339071, -0.644580, -2.822737, -1.245072, 1.570796, 1.909867],accel_mss,speed_ms,0,blend_radius_m)
    |   movel([0.336594, -0.644978, -2.822699, -1.244712, 1.570796, 1.907390],accel_mss,speed_ms,0,blend_radius_m)
    |   movel([0.335177, -0.645740, -2.822626, -1.244023, 1.570796, 1.905973],accel_mss,speed_ms,0,blend_radius_m)
    |   movel([0.333376, -0.647605, -2.822447, -1.242337, 1.570796, 1.904173],accel_mss,speed_ms,0,blend_radius_m)
    |   movel([0.331702, -0.649821, -2.822232, -1.240336, 1.570796, 1.902498],accel_mss,speed_ms,0,blend_radius_m)
    |   movel([0.329626, -0.652327, -2.821986, -1.238075, 1.570796, 1.900422],accel_mss,speed_ms,0,blend_radius_m)
    |   movel([0.327431, -0.654552, -2.821766, -1.236071, 1.570796, 1.898227],accel_mss,speed_ms,0,blend_radius_m)
    |   movel([0.325199, -0.656446, -2.821577, -1.234366, 1.570796, 1.895995],accel_mss,speed_ms,0,blend_radius_m)
    |   movel([0.322999, -0.657965, -2.821425, -1.232999, 1.570796, 1.893796],accel_mss,speed_ms,0,blend_radius_m)
    |   movel([0.320906, -0.659071, -2.821313, -1.232005, 1.570796, 1.891702],accel_mss,speed_ms,0,blend_radius_m)
    |   movel([0.319006, -0.659703, -2.821249, -1.231437, 1.570796, 1.889802],accel_mss,speed_ms,0,blend_radius_m)
    |   movel([0.317365, -0.659836, -2.821235, -1.231318, 1.570796, 1.888161],accel_mss,speed_ms,0,blend_radius_m)
    |   movel([0.316064, -0.659402, -2.821279, -1.231708, 1.570796, 1.886860],accel_mss,speed_ms,0,blend_radius_m)
    |   speed_ms = 0.005
    |   movel([0.316064, -0.652703, -2.814550, -1.245135, 1.570796, 1.886860],accel_mss,speed_ms,0,blend_radius_m)
    |   speed_ms = 0.040
    |   movel([0.297031, -0.681481, -2.811472, -1.219436, 1.570796, 1.867827],accel_mss,speed_ms,0,blend_radius_m)
    |   speed_ms = 0.005
    |   movel([0.297031, -0.688613, -2.818140, -1.205636, 1.570796, 1.867827],accel_mss,speed_ms,0,blend_radius_m)
    |   speed_ms = 0.025
    |   movel([0.292737, -0.713254, -2.815207, -1.183928, 1.570796, 1.863533],accel_mss,speed_ms,0,blend_radius_m)
    |   movel([0.291940, -0.716408, -2.814812, -1.181169, 1.570796, 1.862736],accel_mss,speed_ms,0,blend_radius_m)
    |   movel([0.291178, -0.718063, -2.814603, -1.179723, 1.570796, 1.861975],accel_mss,speed_ms,0,blend_radius_m)
    |   movel([0.290064, -0.719672, -2.814399, -1.178318, 1.570796, 1.860860],accel_mss,speed_ms,0,blend_radius_m)
    |   movel([0.287163, -0.722731, -2.814008, -1.175651, 1.570796, 1.857960],accel_mss,speed_ms,0,blend_radius_m)
    |   movel([0.286186, -0.724523, -2.813776, -1.174090, 1.570796, 1.856982],accel_mss,speed_ms,0,blend_radius_m)
    |   movel([0.285722, -0.726208, -2.813557, -1.172624, 1.570796, 1.856518],accel_mss,speed_ms,0,blend_radius_m)
    |   movel([0.285675, -0.728553, -2.813251, -1.170585, 1.570796, 1.856472],accel_mss,speed_ms,0,blend_radius_m)
    |   movel([0.286255, -0.730443, -2.813002, -1.168944, 1.570796, 1.857051],accel_mss,speed_ms,0,blend_radius_m)
    |   movel([0.287872, -0.733661, -2.812574, -1.166154, 1.570796, 1.858668],accel_mss,speed_ms,0,blend_radius_m)
    |   movel([0.288396, -0.736311, -2.812218, -1.163860, 1.570796, 1.859193],accel_mss,speed_ms,0,blend_radius_m)
    |   movel([0.288528, -0.740579, -2.811638, -1.160172, 1.570796, 1.859324],accel_mss,speed_ms,0,blend_radius_m)
    |   movel([0.288218, -0.742745, -2.811341, -1.158304, 1.570796, 1.859014],accel_mss,speed_ms,0,blend_radius_m)
    |   movel([0.287528, -0.744645, -2.811078, -1.156666, 1.570796, 1.858325],accel_mss,speed_ms,0,blend_radius_m)
    |   movel([0.287013, -0.745418, -2.810970, -1.156001, 1.570796, 1.857810],accel_mss,speed_ms,0,blend_radius_m)
    |   movel([0.286370, -0.746043, -2.810883, -1.155462, 1.570796, 1.857167],accel_mss,speed_ms,0,blend_radius_m)
    |   movel([0.285587, -0.746491, -2.810821, -1.155077, 1.570796, 1.856383],accel_mss,speed_ms,0,blend_radius_m)
    |   movel([0.284653, -0.746727, -2.810788, -1.154874, 1.570796, 1.855450],accel_mss,speed_ms,0,blend_radius_m)
    |   movel([0.284105, -0.748699, -2.810512, -1.153179, 1.570796, 1.854901],accel_mss,speed_ms,0,blend_radius_m)
    |   movel([0.283960, -0.750678, -2.810232, -1.151479, 1.570796, 1.854757],accel_mss,speed_ms,0,blend_radius_m)
    |   movel([0.284532, -0.754504, -2.809687, -1.148198, 1.570796, 1.855329],accel_mss,speed_ms,0,blend_radius_m)
    |   movel([0.285707, -0.757843, -2.809206, -1.145341, 1.570796, 1.856503],accel_mss,speed_ms,0,blend_radius_m)
    |   movel([0.286844, -0.760319, -2.808845, -1.143225, 1.570796, 1.857641],accel_mss,speed_ms,0,blend_radius_m)
    |   movel([0.288585, -0.762570, -2.808515, -1.141304, 1.570796, 1.859382],accel_mss,speed_ms,0,blend_radius_m)
    |   movel([0.290736, -0.764538, -2.808224, -1.139627, 1.570796, 1.861532],accel_mss,speed_ms,0,blend_radius_m)
    |   movel([0.292420, -0.766947, -2.807866, -1.137577, 1.570796, 1.863216],accel_mss,speed_ms,0,blend_radius_m)
    |   movel([0.292816, -0.768530, -2.807628, -1.136230, 1.570796, 1.863613],accel_mss,speed_ms,0,blend_radius_m)
    |   movel([0.292770, -0.770487, -2.807334, -1.134568, 1.570796, 1.863566],accel_mss,speed_ms,0,blend_radius_m)
    |   movel([0.292466, -0.771675, -2.807154, -1.133560, 1.570796, 1.863262],accel_mss,speed_ms,0,blend_radius_m)
    |   movel([0.291884, -0.772966, -2.806957, -1.132465, 1.570796, 1.862681],accel_mss,speed_ms,0,blend_radius_m)
    |   movel([0.291098, -0.774095, -2.806785, -1.131509, 1.570796, 1.861894],accel_mss,speed_ms,0,blend_radius_m)
    |   movel([0.290169, -0.774808, -2.806676, -1.130905, 1.570796, 1.860965],accel_mss,speed_ms,0,blend_radius_m)
    |   movel([0.289526, -0.774882, -2.806665, -1.130842, 1.570796, 1.860322],accel_mss,speed_ms,0,blend_radius_m)
    |   movel([0.289054, -0.774652, -2.806700, -1.131037, 1.570796, 1.859851],accel_mss,speed_ms,0,blend_radius_m)
    |   movel([0.285320, -0.771421, -2.807192, -1.133775, 1.570796, 1.856116],accel_mss,speed_ms,0,blend_radius_m)
    |   movel([0.283748, -0.769440, -2.807492, -1.135457, 1.570796, 1.854545],accel_mss,speed_ms,0,blend_radius_m)
    |   movel([0.282388, -0.767211, -2.807826, -1.137352, 1.570796, 1.853184],accel_mss,speed_ms,0,blend_radius_m)
    |   movel([0.281552, -0.768528, -2.807629, -1.136232, 1.570796, 1.852349],accel_mss,speed_ms,0,blend_radius_m)
    |   movel([0.280945, -0.769840, -2.807431, -1.135117, 1.570796, 1.851742],accel_mss,speed_ms,0,blend_radius_m)
    |   movel([0.280336, -0.772418, -2.807041, -1.132930, 1.570796, 1.851133],accel_mss,speed_ms,0,blend_radius_m)
    |   movel([0.280381, -0.774894, -2.806663, -1.130832, 1.570796, 1.851177],accel_mss,speed_ms,0,blend_radius_m)
    |   movel([0.280920, -0.777209, -2.806307, -1.128873, 1.570796, 1.851716],accel_mss,speed_ms,0,blend_radius_m)
    |   movel([0.282766, -0.781198, -2.805687, -1.125504, 1.570796, 1.853562],accel_mss,speed_ms,0,blend_radius_m)
    |   movel([0.284542, -0.783960, -2.805253, -1.123176, 1.570796, 1.855338],accel_mss,speed_ms,0,blend_radius_m)
    |   movel([0.285038, -0.785149, -2.805065, -1.122174, 1.570796, 1.855834],accel_mss,speed_ms,0,blend_radius_m)
    |   movel([0.285014, -0.785936, -2.804940, -1.121512, 1.570796, 1.855810],accel_mss,speed_ms,0,blend_radius_m)
    |   movel([0.284661, -0.786896, -2.804788, -1.120705, 1.570796, 1.855457],accel_mss,speed_ms,0,blend_radius_m)
    |   movel([0.283980, -0.787944, -2.804621, -1.119824, 1.570796, 1.854777],accel_mss,speed_ms,0,blend_radius_m)
    |   movel([0.283295, -0.788600, -2.804516, -1.119273, 1.570796, 1.854091],accel_mss,speed_ms,0,blend_radius_m)
    |   movel([0.281962, -0.789135, -2.804430, -1.118824, 1.570796, 1.852758],accel_mss,speed_ms,0,blend_radius_m)
    |   movel([0.280166, -0.789628, -2.804351, -1.118410, 1.570796, 1.850963],accel_mss,speed_ms,0,blend_radius_m)
    |   movel([0.279665, -0.790135, -2.804270, -1.117984, 1.570796, 1.850462],accel_mss,speed_ms,0,blend_radius_m)
    |   movel([0.279176, -0.791046, -2.804123, -1.117220, 1.570796, 1.849973],accel_mss,speed_ms,0,blend_radius_m)
    |   movel([0.278930, -0.791993, -2.803970, -1.116426, 1.570796, 1.849726],accel_mss,speed_ms,0,blend_radius_m)
    |   movel([0.278979, -0.793873, -2.803665, -1.114851, 1.570796, 1.849776],accel_mss,speed_ms,0,blend_radius_m)
    |   movel([0.279806, -0.796795, -2.803187, -1.112407, 1.570796, 1.850602],accel_mss,speed_ms,0,blend_radius_m)
    |   movel([0.282019, -0.802536, -2.802236, -1.107617, 1.570796, 1.852816],accel_mss,speed_ms,0,blend_radius_m)
    |   movel([0.284360, -0.808116, -2.801295, -1.102978, 1.570796, 1.855156],accel_mss,speed_ms,0,blend_radius_m)
    |   movel([0.284619, -0.809438, -2.801070, -1.101882, 1.570796, 1.855415],accel_mss,speed_ms,0,blend_radius_m)
    |   movel([0.284546, -0.811022, -2.800798, -1.100569, 1.570796, 1.855342],accel_mss,speed_ms,0,blend_radius_m)
    |   movel([0.283987, -0.812721, -2.800506, -1.099162, 1.570796, 1.854783],accel_mss,speed_ms,0,blend_radius_m)
    |   movel([0.283487, -0.813561, -2.800361, -1.098467, 1.570796, 1.854283],accel_mss,speed_ms,0,blend_radius_m)
    |   movel([0.282096, -0.814998, -2.800112, -1.097279, 1.570796, 1.852892],accel_mss,speed_ms,0,blend_radius_m)
    |   movel([0.281426, -0.815397, -2.800043, -1.096949, 1.570796, 1.852222],accel_mss,speed_ms,0,blend_radius_m)
    |   movel([0.280211, -0.815628, -2.800003, -1.096759, 1.570796, 1.851007],accel_mss,speed_ms,0,blend_radius_m)
    |   movel([0.279193, -0.815306, -2.800058, -1.097024, 1.570796, 1.849990],accel_mss,speed_ms,0,blend_radius_m)
    |   movel([0.278409, -0.814654, -2.800172, -1.097563, 1.570796, 1.849205],accel_mss,speed_ms,0,blend_radius_m)
    |   movel([0.274528, -0.809909, -2.800989, -1.101491, 1.570796, 1.845325],accel_mss,speed_ms,0,blend_radius_m)
    |   movel([0.271008, -0.804718, -2.801870, -1.105801, 1.570796, 1.841804],accel_mss,speed_ms,0,blend_radius_m)
    |   movel([0.267872, -0.799072, -2.802812, -1.110505, 1.570796, 1.838668],accel_mss,speed_ms,0,blend_radius_m)
    |   movel([0.265129, -0.792973, -2.803811, -1.115605, 1.570796, 1.835926],accel_mss,speed_ms,0,blend_radius_m)
    |   movel([0.264285, -0.790532, -2.804206, -1.117651, 1.570796, 1.835081],accel_mss,speed_ms,0,blend_radius_m)
    |   movel([0.263933, -0.787651, -2.804668, -1.120070, 1.570796, 1.834730],accel_mss,speed_ms,0,blend_radius_m)
    |   movel([0.264111, -0.785644, -2.804987, -1.121758, 1.570796, 1.834908],accel_mss,speed_ms,0,blend_radius_m)
    |   movel([0.264533, -0.783475, -2.805330, -1.123584, 1.570796, 1.835330],accel_mss,speed_ms,0,blend_radius_m)
    |   movel([0.265786, -0.778878, -2.806049, -1.127463, 1.570796, 1.836583],accel_mss,speed_ms,0,blend_radius_m)
    |   movel([0.271710, -0.761585, -2.808659, -1.142144, 1.570796, 1.842506],accel_mss,speed_ms,0,blend_radius_m)
    |   movel([0.273050, -0.756811, -2.809355, -1.146223, 1.570796, 1.843846],accel_mss,speed_ms,0,blend_radius_m)
    |   movel([0.273800, -0.752720, -2.809942, -1.149727, 1.570796, 1.844596],accel_mss,speed_ms,0,blend_radius_m)
    |   movel([0.273875, -0.751066, -2.810177, -1.151146, 1.570796, 1.844672],accel_mss,speed_ms,0,blend_radius_m)
    |   movel([0.273697, -0.749755, -2.810363, -1.152271, 1.570796, 1.844493],accel_mss,speed_ms,0,blend_radius_m)
    |   movel([0.273239, -0.748835, -2.810492, -1.153062, 1.570796, 1.844035],accel_mss,speed_ms,0,blend_radius_m)
    |   movel([0.272470, -0.748362, -2.810559, -1.153468, 1.570796, 1.843266],accel_mss,speed_ms,0,blend_radius_m)
    |   movel([0.270671, -0.748274, -2.810571, -1.153543, 1.570796, 1.841467],accel_mss,speed_ms,0,blend_radius_m)
    |   movel([0.269898, -0.748083, -2.810598, -1.153708, 1.570796, 1.840694],accel_mss,speed_ms,0,blend_radius_m)
    |   movel([0.269471, -0.747467, -2.810684, -1.154238, 1.570796, 1.840267],accel_mss,speed_ms,0,blend_radius_m)
    |   movel([0.269732, -0.745748, -2.810925, -1.155717, 1.570796, 1.840528],accel_mss,speed_ms,0,blend_radius_m)
    |   movel([0.270642, -0.743641, -2.811217, -1.157531, 1.570796, 1.841439],accel_mss,speed_ms,0,blend_radius_m)
    |   movel([0.273783, -0.736813, -2.812150, -1.163425, 1.570796, 1.844579],accel_mss,speed_ms,0,blend_radius_m)
    |   movel([0.276622, -0.730070, -2.813051, -1.169268, 1.570796, 1.847419],accel_mss,speed_ms,0,blend_radius_m)
    |   movel([0.279202, -0.723382, -2.813924, -1.175083, 1.570796, 1.849998],accel_mss,speed_ms,0,blend_radius_m)
    |   movel([0.281562, -0.716734, -2.814771, -1.180884, 1.570796, 1.852358],accel_mss,speed_ms,0,blend_radius_m)
    |   movel([0.285832, -0.703469, -2.816403, -1.192517, 1.570796, 1.856629],accel_mss,speed_ms,0,blend_radius_m)
    |   movel([0.289811, -0.690078, -2.817973, -1.204338, 1.570796, 1.860607],accel_mss,speed_ms,0,blend_radius_m)
    |   speed_ms = 0.005
    |   movel([0.289811, -0.682924, -2.811309, -1.218156, 1.570796, 1.860607],accel_mss,speed_ms,0,blend_radius_m)
    |   speed_ms = 0.040
    |   movel([0.275079, -0.717474, -2.807118, -1.187797, 1.570796, 1.845875],accel_mss,speed_ms,0,blend_radius_m)
    |   speed_ms = 0.005
    |   movel([0.275079, -0.725111, -2.813700, -1.173578, 1.570796, 1.845875],accel_mss,speed_ms,0,blend_radius_m)
    |   speed_ms = 0.025
    |   movel([0.268127, -0.734468, -2.812466, -1.165455, 1.570796, 1.838923],accel_mss,speed_ms,0,blend_radius_m)
    |   movel([0.261065, -0.743558, -2.811228, -1.157603, 1.570796, 1.831861],accel_mss,speed_ms,0,blend_radius_m)
    |   movel([0.253905, -0.752376, -2.809991, -1.150022, 1.570796, 1.824701],accel_mss,speed_ms,0,blend_radius_m)
    |   movel([0.246668, -0.760894, -2.808761, -1.142734, 1.570796, 1.817465],accel_mss,speed_ms,0,blend_radius_m)
    |   movel([0.252354, -0.752210, -2.810015, -1.150164, 1.570796, 1.823151],accel_mss,speed_ms,0,blend_radius_m)
    |   movel([0.257714, -0.743342, -2.811258, -1.157788, 1.570796, 1.828511],accel_mss,speed_ms,0,blend_radius_m)
    |   movel([0.262708, -0.734350, -2.812482, -1.165558, 1.570796, 1.833504],accel_mss,speed_ms,0,blend_radius_m)
    |   movel([0.267297, -0.725292, -2.813677, -1.173421, 1.570796, 1.838093],accel_mss,speed_ms,0,blend_radius_m)
    |   movel([0.261463, -0.732979, -2.812665, -1.166745, 1.570796, 1.832260],accel_mss,speed_ms,0,blend_radius_m)
    |   movel([0.255548, -0.740463, -2.811654, -1.160272, 1.570796, 1.826345],accel_mss,speed_ms,0,blend_radius_m)
    |   movel([0.249550, -0.747743, -2.810646, -1.154000, 1.570796, 1.820347],accel_mss,speed_ms,0,blend_radius_m)
    |   movel([0.243487, -0.754796, -2.809645, -1.147948, 1.570796, 1.814283],accel_mss,speed_ms,0,blend_radius_m)
    |   movel([0.236727, -0.762462, -2.808531, -1.141396, 1.570796, 1.807524],accel_mss,speed_ms,0,blend_radius_m)
    |   movel([0.230254, -0.770278, -2.807365, -1.134746, 1.570796, 1.801050],accel_mss,speed_ms,0,blend_radius_m)
    |   movel([0.227253, -0.774365, -2.806744, -1.131280, 1.570796, 1.798049],accel_mss,speed_ms,0,blend_radius_m)
    |   movel([0.224534, -0.778541, -2.806101, -1.127747, 1.570796, 1.795330],accel_mss,speed_ms,0,blend_radius_m)
    |   movel([0.222241, -0.782708, -2.805450, -1.124231, 1.570796, 1.793037],accel_mss,speed_ms,0,blend_radius_m)
    |   movel([0.220493, -0.786767, -2.804808, -1.120814, 1.570796, 1.791290],accel_mss,speed_ms,0,blend_radius_m)
    |   movel([0.221810, -0.782059, -2.805552, -1.124778, 1.570796, 1.792606],accel_mss,speed_ms,0,blend_radius_m)
    |   movel([0.223499, -0.777060, -2.806330, -1.128999, 1.570796, 1.794295],accel_mss,speed_ms,0,blend_radius_m)
    |   movel([0.225535, -0.771834, -2.807130, -1.133425, 1.570796, 1.796331],accel_mss,speed_ms,0,blend_radius_m)
    |   movel([0.227887, -0.766443, -2.807941, -1.138005, 1.570796, 1.798683],accel_mss,speed_ms,0,blend_radius_m)
    |   movel([0.230522, -0.760956, -2.808752, -1.142681, 1.570796, 1.801319],accel_mss,speed_ms,0,blend_radius_m)
    |   movel([0.233414, -0.755437, -2.809553, -1.147399, 1.570796, 1.804210],accel_mss,speed_ms,0,blend_radius_m)
    |   movel([0.236525, -0.749959, -2.810334, -1.152096, 1.570796, 1.807321],accel_mss,speed_ms,0,blend_radius_m)
    |   movel([0.239819, -0.744599, -2.811084, -1.156706, 1.570796, 1.810616],accel_mss,speed_ms,0,blend_radius_m)
    |   movel([0.233910, -0.753009, -2.809901, -1.149479, 1.570796, 1.804707],accel_mss,speed_ms,0,blend_radius_m)
    |   movel([0.228354, -0.761414, -2.808685, -1.142290, 1.570796, 1.799150],accel_mss,speed_ms,0,blend_radius_m)
    |   movel([0.223129, -0.769788, -2.807439, -1.135162, 1.570796, 1.793925],accel_mss,speed_ms,0,blend_radius_m)
    |   movel([0.218214, -0.778107, -2.806168, -1.128114, 1.570796, 1.789011],accel_mss,speed_ms,0,blend_radius_m)
    |   movel([0.213595, -0.786341, -2.804876, -1.121172, 1.570796, 1.784391],accel_mss,speed_ms,0,blend_radius_m)
    |   movel([0.209243, -0.794472, -2.803567, -1.114349, 1.570796, 1.780039],accel_mss,speed_ms,0,blend_radius_m)
    |   movel([0.201260, -0.810334, -2.800916, -1.101139, 1.570796, 1.772056],accel_mss,speed_ms,0,blend_radius_m)
    |   movel([0.203464, -0.804990, -2.801824, -1.105575, 1.570796, 1.774260],accel_mss,speed_ms,0,blend_radius_m)
    |   movel([0.205242, -0.799405, -2.802757, -1.110227, 1.570796, 1.776038],accel_mss,speed_ms,0,blend_radius_m)
    |   movel([0.208401, -0.788563, -2.804522, -1.119304, 1.570796, 1.779197],accel_mss,speed_ms,0,blend_radius_m)
    |   movel([0.210178, -0.783603, -2.805310, -1.123477, 1.570796, 1.780974],accel_mss,speed_ms,0,blend_radius_m)
    |   movel([0.212078, -0.779038, -2.806024, -1.127327, 1.570796, 1.782875],accel_mss,speed_ms,0,blend_radius_m)
    |   movel([0.216697, -0.769406, -2.807497, -1.135486, 1.570796, 1.787493],accel_mss,speed_ms,0,blend_radius_m)
    |   movel([0.215720, -0.770822, -2.807283, -1.134284, 1.570796, 1.786517],accel_mss,speed_ms,0,blend_radius_m)
    |   movel([0.214075, -0.772682, -2.807001, -1.132706, 1.570796, 1.784871],accel_mss,speed_ms,0,blend_radius_m)
    |   movel([0.204895, -0.781667, -2.805614, -1.125108, 1.570796, 1.775691],accel_mss,speed_ms,0,blend_radius_m)
    |   movel([0.201596, -0.785073, -2.805077, -1.122238, 1.570796, 1.772393],accel_mss,speed_ms,0,blend_radius_m)
    |   movel([0.197922, -0.789844, -2.804316, -1.118228, 1.570796, 1.768719],accel_mss,speed_ms,0,blend_radius_m)
    |   movel([0.194516, -0.794881, -2.803500, -1.114007, 1.570796, 1.765312],accel_mss,speed_ms,0,blend_radius_m)
    |   movel([0.188382, -0.804981, -2.801825, -1.105583, 1.570796, 1.759178],accel_mss,speed_ms,0,blend_radius_m)
    |   movel([0.190795, -0.799774, -2.802695, -1.109919, 1.570796, 1.761591],accel_mss,speed_ms,0,blend_radius_m)
    |   movel([0.192889, -0.794595, -2.803547, -1.114247, 1.570796, 1.763685],accel_mss,speed_ms,0,blend_radius_m)
    |   movel([0.197009, -0.784152, -2.805223, -1.123014, 1.570796, 1.767806],accel_mss,speed_ms,0,blend_radius_m)
    |   movel([0.199573, -0.778593, -2.806093, -1.127703, 1.570796, 1.770370],accel_mss,speed_ms,0,blend_radius_m)
    |   movel([0.202507, -0.772907, -2.806967, -1.132515, 1.570796, 1.773304],accel_mss,speed_ms,0,blend_radius_m)
    |   movel([0.209227, -0.761221, -2.808713, -1.142455, 1.570796, 1.780023],accel_mss,speed_ms,0,blend_radius_m)
    |   movel([0.223920, -0.737541, -2.812052, -1.162796, 1.570796, 1.794717],accel_mss,speed_ms,0,blend_radius_m)
    |   movel([0.218305, -0.742455, -2.811381, -1.158554, 1.570796, 1.789101],accel_mss,speed_ms,0,blend_radius_m)
    |   movel([0.212782, -0.747691, -2.810653, -1.154045, 1.570796, 1.783579],accel_mss,speed_ms,0,blend_radius_m)
    |   movel([0.207379, -0.753202, -2.809873, -1.149313, 1.570796, 1.778176],accel_mss,speed_ms,0,blend_radius_m)
    |   movel([0.202138, -0.758944, -2.809046, -1.144399, 1.570796, 1.772934],accel_mss,speed_ms,0,blend_radius_m)
    |   movel([0.197095, -0.764873, -2.808174, -1.139342, 1.570796, 1.767892],accel_mss,speed_ms,0,blend_radius_m)
    |   movel([0.192276, -0.770955, -2.807263, -1.134171, 1.570796, 1.763072],accel_mss,speed_ms,0,blend_radius_m)
    |   movel([0.187710, -0.777142, -2.806317, -1.128930, 1.570796, 1.758507],accel_mss,speed_ms,0,blend_radius_m)
    |   movel([0.183429, -0.783402, -2.805341, -1.123646, 1.570796, 1.754226],accel_mss,speed_ms,0,blend_radius_m)
    |   movel([0.184563, -0.781502, -2.805639, -1.125248, 1.570796, 1.755359],accel_mss,speed_ms,0,blend_radius_m)
    |   movel([0.185626, -0.779401, -2.805967, -1.127021, 1.570796, 1.756423],accel_mss,speed_ms,0,blend_radius_m)
    |   movel([0.187595, -0.774841, -2.806671, -1.130876, 1.570796, 1.758391],accel_mss,speed_ms,0,blend_radius_m)
    |   movel([0.191200, -0.766084, -2.807994, -1.138311, 1.570796, 1.761996],accel_mss,speed_ms,0,blend_radius_m)
    |   movel([0.194972, -0.758401, -2.809124, -1.144864, 1.570796, 1.765769],accel_mss,speed_ms,0,blend_radius_m)
    |   movel([0.199027, -0.750653, -2.810236, -1.151500, 1.570796, 1.769823],accel_mss,speed_ms,0,blend_radius_m)
    |   movel([0.203355, -0.742843, -2.811327, -1.158219, 1.570796, 1.774151],accel_mss,speed_ms,0,blend_radius_m)
    |   movel([0.207941, -0.734972, -2.812398, -1.165019, 1.570796, 1.778737],accel_mss,speed_ms,0,blend_radius_m)
    |   movel([0.212779, -0.727027, -2.813451, -1.171911, 1.570796, 1.783576],accel_mss,speed_ms,0,blend_radius_m)
    |   movel([0.217863, -0.719015, -2.814483, -1.178891, 1.570796, 1.788659],accel_mss,speed_ms,0,blend_radius_m)
    |   movel([0.228720, -0.702753, -2.816489, -1.193146, 1.570796, 1.799517],accel_mss,speed_ms,0,blend_radius_m)
    |   movel([0.224218, -0.707892, -2.815868, -1.188629, 1.570796, 1.795015],accel_mss,speed_ms,0,blend_radius_m)
    |   movel([0.210460, -0.722428, -2.814047, -1.175915, 1.570796, 1.781257],accel_mss,speed_ms,0,blend_radius_m)
    |   movel([0.205971, -0.727360, -2.813407, -1.171622, 1.570796, 1.776768],accel_mss,speed_ms,0,blend_radius_m)
    |   movel([0.201658, -0.732479, -2.812732, -1.167178, 1.570796, 1.772454],accel_mss,speed_ms,0,blend_radius_m)
    |   movel([0.197675, -0.737759, -2.812022, -1.162608, 1.570796, 1.768471],accel_mss,speed_ms,0,blend_radius_m)
    |   movel([0.194163, -0.743189, -2.811279, -1.157921, 1.570796, 1.764959],accel_mss,speed_ms,0,blend_radius_m)
    |   movel([0.198947, -0.734314, -2.812487, -1.165588, 1.570796, 1.769744],accel_mss,speed_ms,0,blend_radius_m)
